(* IEC 61131-3 sources: elnaProjects/ElpcLogic/PomarKc7Changed/build_USO_ecl/_ (part 6) *)

  StrAlg.CanRun := StrAlg.inCanRun;
  StrAlg.OpcCommandsDisabled := StrAlg.inOpcCommandsDisabled;

  IF StrAlg.isRuning THEN

      StrAlg.hasError := kran3bOpen.error OR kran4Open.error OR kran5Close.error OR kran5Close.error
      OR kran1Open.error OR kran2Open.error OR kran3bClose.error OR kran4Close.error OR testUnsuccessfulFilling.error;

      IF kran4Open.top THEN
          runPhase(waitAfterKran4);
      END_IF;

      IF waitAfterKran4.top THEN
          runPhase(kran5Close);
      END_IF;

      IF kran3bOpen.top AND kran5Close.top THEN
         runPhase(waitAfterKran5);
         runPhase(didPKran1);
      END_IF;

      (*IF didPKran1.start AND NOT didPKran1.top THEN
      didPKran1.top:= im.singleSignals.dP_gazgaz_Kran1.Q;
      END_IF;*)

      IF waitAfterKran5.top AND didPKran1.top THEN
            runPhase(kran1Open);
  	runPhase(kran2Open);
      END_IF;

      IF kran1Open.top AND kran2Open.top THEN
            runPhase(kran4Close);
  	runPhase(kran3bClose);
      END_IF;

      IF kran4Close.top AND kran3bClose.top THEN

            runPhase(RunProtection_kr1);
            runPhase(RunProtection_kr2);

            (*runAiProtection(protections.Pgaza_na_vhode_nagnetatelia);
            runAiProtection(protections.Pgaza_na_vhode_nagnetatelia);
            runAiProtection(protections.Pgaza_na_vyhode_nagnetatelia);
            runAiProtection(protections.dPmaslo_gaz);
            runAiProtection(protections.Pmaslo_sm_nizkoe);
            runAiProtection(protections.Pmaslo_sm_vysokoe);*)

      END_IF;

      IF BreakPuskTimer.top AND NOT (RunProtection_kr1.top AND RunProtection_kr2.top ) THEN
  	testUnsuccessfulFilling.error:=TRUE;
      END_IF;

      IF RunProtection_kr1.top AND RunProtection_kr2.top THEN
            resetPhase(BreakPuskTimer);
  	waitReset(IN:=TRUE, PT:= T#2S);
      END_IF;

      IF waitReset.Q AND NOT (algoritms.Apusk.isRuning OR algoritms.SemiAutoPusk.isRuning) THEN
  	resetIfRunning(StrAlg);
      END_IF;

      StrAlg.isEnded:= RunProtection_kr1.top AND RunProtection_kr2.top;
  END_IF;

  StrAlg.CanRun := StrAlg.inCanRun;
  StrAlg.OpcCommandsDisabled := StrAlg.inOpcCommandsDisabled;

  (* ---- Если управление с ВУ заблокировано, то  передаем команду из алгоритма ---- *)
  IF StrAlg.inOpcCommandsDisabled THEN
  	StrAlg.inCommand := StrAlg.inCommand_Alg;
  ELSE (* иначе передаем команду с АРМа*)
  	StrAlg.inCommand := StrAlg.inCommand_ARM;
  END_IF;

  _sunpackerCommand(command := StrAlg.inCommand);
  	source := _sunpackerCommand.source;
  	cmd := _sunpackerCommand.cmd;

  IF cmd <> 0 AND lastCmd <> cmd AND (((NOT StrAlg.opcCommandsDisabled) AND source > 0) OR source = 0) then
  	CASE BYTE_TO_INT(cmd) OF
  		(*cmdRun*) 1: 	IF (StrAlg.CanRun) THEN
  					StrAlg.isRuning := TRUE;
  					StrAlg.isEnded := FALSE;
  					StrAlg.hasError := FALSE;
  					(*****************       OnRun       *****************)

                                                    runPhase(kran3bOpen);
                                                    runPhase(kran4Open);
                                                    runPhase(BreakPuskTimer);
                                                    runPhase(testUnsuccessfulFilling);

  					cmd_for_Status := cmd;
  					source_for_Status := source;
  					command_error_for_Status := 0;
  				ELSE
  					StrAlg.isRuning := FALSE;
  					StrAlg.isEnded := FALSE;
  					StrAlg.hasError 	:= FALSE;

  					cmd_for_Status := 0;
  					source_for_Status := source;
  					command_error_for_Status := cmd;
  				END_IF;
  		(*cmdReset*) 2: 	StrAlg.isRuning := FALSE;
  				StrAlg.isEnded := FALSE;
  				StrAlg.hasError 	:= FALSE;

                                           (*****************       OnReset       *****************)
                                          StrAlg.inCanRun:=FALSE;
                                          waitReset(IN:=FALSE);

                                          resetPhase(BreakPuskTimer);
                                          resetPhase(kran3bOpen);
                                          resetPhase(kran4Open);
                                          resetPhase(waitAfterKran4);
                                          resetPhase(kran5Close);
                                          resetPhase(didPKran1);
                                          resetPhase(kran1Open);
                                          resetPhase(kran2Open);
                                          resetPhase(kran3bClose);
                                          resetPhase(kran4Close);
  	                              resetPhase(RunProtection_kr1);
                                          resetPhase(RunProtection_kr2);
                                          resetPhase(waitAfterKran5);
                                          resetPhase(testUnsuccessfulFilling);

  				cmd_for_Status := cmd;
  				source_for_Status := source;
  				command_error_for_Status := 0;
  	END_CASE;
  	resetCmdTimer(IN := false);
  	resetCmdTimerPriznak := TRUE;
  END_IF;
  lastCmd := cmd;

  resetCmdTimer(IN := resetCmdTimerPriznak, PT := T#5S);
  IF resetCmdTimer.Q THEN
  	resetCmdTimerPriznak := FALSE;
  	source_for_Status := 0;
  	cmd_for_Status := 0;
  	command_error_for_Status := 0;
  END_IF;

  StrAlg.Start:= BreakPuskTimer.startStatus
              OR kran3bOpen.startStatus
              OR kran4Open.startStatus
              OR waitAfterKran4.startStatus
              OR kran5Close.startStatus
              OR didPKran1.startStatus
              OR kran1Open.startStatus
              OR kran2Open.startStatus
              OR kran3bClose.startStatus
              OR kran4Close.startStatus
              OR RunProtection_kr1.startStatus
              OR RunProtection_kr2.startStatus
              OR waitAfterKran5.startStatus
              OR testUnsuccessfulFilling.startStatus;

  StrAlg.Error:= BreakPuskTimer.errorStatus
              OR kran3bOpen.errorStatus
              OR kran4Open.errorStatus
              OR waitAfterKran4.errorStatus
              OR kran5Close.errorStatus
              OR didPKran1.errorStatus
              OR kran1Open.errorStatus
              OR kran2Open.errorStatus
              OR kran3bClose.errorStatus
              OR kran4Close.errorStatus
              OR RunProtection_kr1.errorStatus
              OR RunProtection_kr2.errorStatus
              OR waitAfterKran5.errorStatus
              OR testUnsuccessfulFilling.errorStatus;

  StrAlg.Top:=   BreakPuskTimer.topStatus
              OR kran3bOpen.topStatus
              OR kran4Open.topStatus
              OR waitAfterKran4.topStatus
              OR kran5Close.topStatus
              OR didPKran1.topStatus
              OR kran1Open.topStatus
              OR kran2Open.topStatus
              OR kran3bClose.topStatus
              OR kran4Close.topStatus
              OR RunProtection_kr1.topStatus
              OR RunProtection_kr2.topStatus
              OR waitAfterKran5.topStatus
              OR testUnsuccessfulFilling.topStatus;

  (*TODO: TYPE PROGRAM CODE HERE*)
  StrAlg.status :=  SHL(BYTE_TO_DWORD(source_for_Status), 29)
  			OR SHL(BYTE_TO_DWORD(cmd_for_Status), 26)
  			OR SHL(BYTE_TO_DWORD(command_error_for_Status), 23)
  			OR SHL(BOOL_TO_DWORD(StrAlg.OpcCommandsDisabled ), 21)
  			OR SHL(BOOL_TO_DWORD(StrAlg.hasError),4)
  			OR SHL(BOOL_TO_DWORD(StrAlg.CanRun),2)
  			OR SHL(BOOL_TO_DWORD(StrAlg.isEnded),1)
  			OR BOOL_TO_DWORD(StrAlg.isRuning);
END_FUNCTION_BLOCK

FUNCTION_BLOCK engineRunAlg
  VAR_IN_OUT
    StrAlg : struct_Alg;
  END_VAR
  VAR
    BreakPuskTimer : struct_PhaseAlgoritm;
    RunProtection_mvoff : struct_PhaseAlgoritm;
    LowOil_upStopust : struct_PhaseAlgoritm;
    mvOn : struct_PhaseAlgoritm;
    AutoPns_ph : struct_PhaseAlgoritm;
    AutoAvom_ph : struct_PhaseAlgoritm;
    pnsOff : struct_PhaseAlgoritm;
    testUnsuccessful : struct_PhaseAlgoritm;
    fb_BreakPuskTimer : fb_ph_Timer;
    fb_RunProtection_mvoff : fb_ph_DIprotection;
    fb_LowOil_upStopust : fb_ph_WaitAnalogValue;
    fb_mvOn : fb_ph_SectionSwitch;
    fb_AutoPns_ph : fb_ph_algoritm;
    fb_AutoAvom_ph : fb_ph_algoritm;
    fb_pnsOff : fb_ph_Switch;
    fb_testUnsuccessful : fb_ph_CustomPhase;
    _sunpackerCommand : fb_sunpackerCommand;
    _DualStateImAction : TYPE_DualStateImAction;
    _PhaseAlgoritmAction : TYPE_PhaseAlgoritmAction;
    source : BYTE;
    cmd : BYTE;
    lastCmd : BYTE;
    source_for_Status : BYTE;
    cmd_for_Status : BYTE;
    command_error_for_Status : BYTE;
    resetCmdTimer : TON;
    resetCmdTimerPriznak : BOOL;
    onInit : BOOL;
    waitReset : TON;
  END_VAR
  VAR_EXTERNAL
    IM : ImConfig;
    algoritms : AlgoritmsConfig;
    ai : AiConfig;
    protections : ProtectionsConfig;
    AlgTimers : struct_AlgTimers;
  END_VAR

  IF NOT onInit THEN

       fb_BreakPuskTimer(phaseNumber:=0, delay:=T#665S);
     fb_LowOil_upStopust(phaseNumber:=1);
                 fb_mvOn(phaseNumber:=2, act:=_on);
           fb_AutoPns_ph(phaseNumber:=3, act:=_run, waitCompletion:=FALSE);
          fb_AutoAvom_ph(phaseNumber:=4, act:=_run, waitCompletion:=FALSE);
               fb_pnsOff(phaseNumber:=5, act:=_off);
  fb_RunProtection_mvoff(phaseNumber:=7, act:=_run);
     fb_testUnsuccessful(phaseNumber:=17);

  onInit:=TRUE;
  END_IF;

          fb_BreakPuskTimer(StrPh:=BreakPuskTimer, timer:=AlgTimers.engineRun_BreakPuskTimer);
       (* fb_LowOil_upStopust(StrPh:=LowOil_upStopust, ai:=ai.Pmasla_posle_GNS, more:=im.AutoPns_UstStop.Value);*)
                    fb_mvOn(StrPh:=mvOn, Im:=Im.mv);
              fb_AutoPns_ph(StrPh:=AutoPns_ph, alg:=algoritms.AutoPns);
             fb_AutoAvom_ph(StrPh:=AutoAvom_ph, alg:=algoritms.AutoAvom);
                  fb_pnsOff(StrPh:=pnsOff, Im:=Im.pns);
    (*fb_RunProtection_mvoff(StrPh:=RunProtection_mvoff, StrDiP:=protections.Pgaza_na_vyhode_nagnetatelia_GPA_STOP);*)
        fb_testUnsuccessful(StrPh:=testUnsuccessful);

  StrAlg.CanRun := StrAlg.inCanRun;
  StrAlg.OpcCommandsDisabled := StrAlg.inOpcCommandsDisabled;

  IF StrAlg.isRuning THEN

      StrAlg.hasError := mvOn.error OR pnsOff.error OR testUnsuccessful.error;

      IF mvOn.top THEN
          runPhase(RunProtection_mvoff);
          runPhase(AutoAvom_ph);
          runPhase(LowOil_upStopust);
      END_IF;
      (*
      IF AutoAvom_ph.top THEN
          algoritms.AutoAvom.inOpcCommandsDisabled:=FALSE;
      END_IF;
      *)
      IF LowOil_upStopust.top THEN
          runPhase(pnsOff);
      END_IF;

      IF pnsOff.top THEN
         runPhase(AutoPns_ph);
      END_IF;

      IF BreakPuskTimer.top AND NOT AutoPns_ph.top THEN
            testUnsuccessful.error:=TRUE;
      END_IF;

      IF AutoPns_ph.top THEN
            resetPhase(BreakPuskTimer);
  	waitReset(IN:=TRUE, PT:= T#2S);
      END_IF;

      IF waitReset.Q AND NOT (algoritms.Apusk.isRuning OR algoritms.SemiAutoPusk.isRuning) THEN
  	resetIfRunning(StrAlg);
      END_IF;

      StrAlg.isEnded:= AutoPns_ph.top;
  END_IF;

  StrAlg.CanRun := StrAlg.inCanRun;
  StrAlg.OpcCommandsDisabled := StrAlg.inOpcCommandsDisabled;

  (* ---- Если управление с ВУ заблокировано, то  передаем команду из алгоритма ---- *)
  IF StrAlg.inOpcCommandsDisabled THEN
  	StrAlg.inCommand := StrAlg.inCommand_Alg;
  ELSE (* иначе передаем команду с АРМа*)
  	StrAlg.inCommand := StrAlg.inCommand_ARM;
  END_IF;

  _sunpackerCommand(command := StrAlg.inCommand);
  	source := _sunpackerCommand.source;
  	cmd := _sunpackerCommand.cmd;

  IF cmd <> 0 AND lastCmd <> cmd AND (((NOT StrAlg.opcCommandsDisabled) AND source > 0) OR source = 0) then
  	CASE BYTE_TO_INT(cmd) OF
  		(*cmdRun*) 1: 	IF (StrAlg.CanRun) THEN
  					StrAlg.isRuning := TRUE;
  					StrAlg.isEnded := FALSE;
  					StrAlg.hasError := FALSE;
  					(*****************       OnRun       *****************)

                                                    runPhase(mvOn);
                                                    runPhase(BreakPuskTimer);
                                                    runPhase(testUnsuccessful);

  					cmd_for_Status := cmd;
  					source_for_Status := source;
  					command_error_for_Status := 0;
  				ELSE
  					StrAlg.isRuning := FALSE;
  					StrAlg.isEnded := FALSE;
  					StrAlg.hasError 	:= FALSE;

  					cmd_for_Status := 0;
  					source_for_Status := source;
  					command_error_for_Status := cmd;
  				END_IF;
  		(*cmdReset*) 2: 	StrAlg.isRuning := FALSE;
  				StrAlg.isEnded := FALSE;
  				StrAlg.hasError 	:= FALSE;

                                           (*****************       OnReset       *****************)
                                          StrAlg.inCanRun:=FALSE;
                                          waitReset(IN:=FALSE);

                                          resetPhase(BreakPuskTimer);
                                          resetPhase(RunProtection_mvoff);
                                          resetPhase(LowOil_upStopust);
                                          resetPhase(mvOn);
                                          resetPhase(AutoPns_ph);
                                          resetPhase(AutoAvom_ph);
                                          resetPhase(pnsOff);
                                          resetPhase(testUnsuccessful);

  				cmd_for_Status := cmd;
  				source_for_Status := source;
  				command_error_for_Status := 0;
  	END_CASE;
  	resetCmdTimer(IN := false);
  	resetCmdTimerPriznak := TRUE;
  END_IF;
  lastCmd := cmd;

  resetCmdTimer(IN := resetCmdTimerPriznak, PT := T#5S);
  IF resetCmdTimer.Q THEN
  	resetCmdTimerPriznak := FALSE;
  	source_for_Status := 0;
  	cmd_for_Status := 0;
  	command_error_for_Status := 0;
  END_IF;

  StrAlg.Start:= BreakPuskTimer.startStatus
              OR RunProtection_mvoff.startStatus
              OR LowOil_upStopust.startStatus
              OR mvOn.startStatus
              OR AutoPns_ph.startStatus
              OR AutoAvom_ph.startStatus
              OR pnsOff.startStatus
              OR testUnsuccessful.startStatus;

  StrAlg.Error:= BreakPuskTimer.errorStatus
              OR RunProtection_mvoff.errorStatus
              OR LowOil_upStopust.errorStatus
              OR mvOn.errorStatus
              OR AutoPns_ph.errorStatus
              OR AutoAvom_ph.errorStatus
              OR pnsOff.errorStatus
              OR testUnsuccessful.errorStatus;

  StrAlg.Top:=   BreakPuskTimer.topStatus
              OR RunProtection_mvoff.topStatus
              OR LowOil_upStopust.topStatus
              OR mvOn.topStatus
              OR AutoPns_ph.topStatus
              OR AutoAvom_ph.topStatus
              OR pnsOff.topStatus
              OR testUnsuccessful.topStatus;

  (*TODO: TYPE PROGRAM CODE HERE*)
  StrAlg.status :=  SHL(BYTE_TO_DWORD(source_for_Status), 29)
  			OR SHL(BYTE_TO_DWORD(cmd_for_Status), 26)
  			OR SHL(BYTE_TO_DWORD(command_error_for_Status), 23)
  			OR SHL(BOOL_TO_DWORD(StrAlg.OpcCommandsDisabled ), 21)
  			OR SHL(BOOL_TO_DWORD(StrAlg.hasError),4)
  			OR SHL(BOOL_TO_DWORD(StrAlg.CanRun),2)
  			OR SHL(BOOL_TO_DWORD(StrAlg.isEnded),1)
  			OR BOOL_TO_DWORD(StrAlg.isRuning);
END_FUNCTION_BLOCK

FUNCTION_BLOCK puskKalg
  VAR_IN_OUT
    StrAlg : struct_Alg;
  END_VAR
  VAR
    puskOilSystem : struct_PhaseAlgoritm;
  END_VAR
  VAR_IN_OUT
    questionFilling : struct_Question;
  END_VAR
  VAR
    filling : struct_PhaseAlgoritm;
  END_VAR
  VAR_IN_OUT
    questionUnload : struct_Question;
  END_VAR
  VAR
    kran3bOpen : struct_PhaseAlgoritm;
    kran4Close : struct_PhaseAlgoritm;
    kran1Close : struct_PhaseAlgoritm;
    kran2Close : struct_PhaseAlgoritm;
    kran5open : struct_PhaseAlgoritm;
    wait720 : struct_PhaseAlgoritm;
    noGasInPipe : struct_PhaseAlgoritm;
    AutoNUoff : struct_PhaseAlgoritm;
    nu1Off : struct_PhaseAlgoritm;
    nu2Off : struct_PhaseAlgoritm;
    pnsWaitOff : struct_PhaseAlgoritm;
    testUnsuccessfulUnfill : struct_PhaseAlgoritm;
    fb_puskOilSystem : fb_ph_algoritm;
    fb_questionFilling : fb_Question;
    fb_filling : fb_ph_algoritm;
    fb_questionUnload : fb_Question;
    fb_kran3bOpen : fb_ph_Kran;
    fb_kran4Close : fb_ph_CustomPhase;
    fb_kran1Close : fb_ph_Kran;
    fb_kran2Close : fb_ph_Kran;
    fb_kran5open : fb_ph_Kran;
    fb_wait720 : fb_ph_Timer;
    fb_noGasInPipe : fb_ph_CustomPhase;
    fb_AutoNUoff : fb_ph_algoritm;
    fb_nu1Off : fb_ph_OilPump;
    fb_nu2Off : fb_ph_OilPump;
    fb_pnsWaitOff : fb_ph_algoritm;
    fb_testUnsuccessfulUnfill : fb_ph_CustomPhase;
    _sunpackerCommand : fb_sunpackerCommand;
    _DualStateImAction : TYPE_DualStateImAction;
    _Answers : TYPE_Answers;
    _statusDualInput : TYPE_statusDualInput;
    _StatusAi : TYPE_StatusAi;
    _PhaseAlgoritmAction : TYPE_PhaseAlgoritmAction;
    source : BYTE;
    cmd : BYTE;
    lastCmd : BYTE;
    source_for_Status : BYTE;
    cmd_for_Status : BYTE;
    command_error_for_Status : BYTE;
    resetCmdTimer : TON;
    resetCmdTimerPriznak : BOOL;
    OpcCommandsKransEnabled : BOOL;
    OpcCommandsKransDisabled : BOOL;
    _resetQuestion1 : BOOL;
    _resetQuestion2 : BOOL;
    onInit : BOOL;
    waitReset : TON;
  END_VAR
  VAR_EXTERNAL
    IM : ImConfig;
    algoritms : AlgoritmsConfig;
    ai : AiConfig;
    AlgTimers : struct_AlgTimers;
    ModeGpa : TYPE_ModeGpa;
    algManager : struct_AlgoritmsManager;
    protections : ProtectionsConfig;
  END_VAR
  VAR CONSTANT
    Ust_Pgaza : LREAL      := 0.3;
  END_VAR

  IF NOT onInit THEN

            fb_puskOilSystem(phaseNumber:=0, act:=_run, waitCompletion:=TRUE);
        questionFilling.AnswerVariants:=_Answers.ANS_YES;
                  fb_filling(phaseNumber:=1, act:=_run, waitCompletion:=TRUE);
      questionUnload.AnswerVariants:=_Answers.ANS_YES;
               fb_kran3bOpen(phaseNumber:=3, act:=_on);
               fb_kran4Close(phaseNumber:=4);
               fb_kran1Close(phaseNumber:=5, act:=_off);
               fb_kran2Close(phaseNumber:=6, act:=_off);
                fb_kran5open(phaseNumber:=7, act:=_on);
                  fb_wait720(phaseNumber:=8, delay:=T#720S);
              fb_noGasInPipe(phaseNumber:=9);
                fb_AutoNUoff(phaseNumber:=10, act:=_reset, waitCompletion:=FALSE);
                   fb_nu1Off(phaseNumber:=11, act:=_off);
                   fb_nu2Off(phaseNumber:=12, act:=_off);
               fb_pnsWaitOff(phaseNumber:=15, act:=_run, waitCompletion:=TRUE);
   fb_testUnsuccessfulUnfill(phaseNumber:=18);

  onInit:=TRUE;
  END_IF;

            fb_puskOilSystem(StrPh:=puskOilSystem, alg:=algoritms.puskOilSystem);
          fb_questionFilling(StrQ:=questionFilling);
                  fb_filling(StrPh:=filling, alg:=algoritms.filling);
           fb_questionUnload(StrQ:=questionUnload);
               fb_kran3bOpen(StrPh:=kran3bOpen, Im:=Im.kran3b);
               fb_kran4Close(StrPh:=kran4Close);
               fb_kran1Close(StrPh:=kran1Close, Im:=Im.kran1);
               fb_kran2Close(StrPh:=kran2Close, Im:=Im.kran2);
                fb_kran5open(StrPh:=kran5open, Im:=Im.kran5);
                  fb_wait720(StrPh:=wait720, timer:=AlgTimers.puskK_wait720);
              fb_noGasInPipe(StrPh:=noGasInPipe);
                fb_AutoNUoff(StrPh:=AutoNUoff, alg:=algoritms.autoNu);
                   fb_nu1Off(StrPh:=nu1Off, Im:=Im.nu1);
                   fb_nu2Off(StrPh:=nu2Off, Im:=Im.nu2);
               fb_pnsWaitOff(StrPh:=pnsWaitOff, alg:=algoritms.vibegPNS);
   fb_testUnsuccessfulUnfill(StrPh:=testUnsuccessfulUnfill);

  StrAlg.CanRun := StrAlg.inCanRun;
  StrAlg.OpcCommandsDisabled := StrAlg.inOpcCommandsDisabled;

  IF StrAlg.isRuning THEN

      StrAlg.hasError := kran3bOpen.error OR kran1Close.error OR kran2Close.error OR kran5open.error OR testUnsuccessfulUnfill.error;

      IF puskOilSystem.top THEN
           IF NOT _resetQuestion1 THEN
           askQuestion(questionFilling);
           _resetQuestion1:=TRUE;
           END_IF;
      END_IF;

      IF questionFilling.answer = _Answers.ANS_YES THEN
          runPhase(filling);
          resetQuestion(questionFilling);
      END_IF;

      IF filling.top THEN
         OpcCommandsKransEnabled:=TRUE;
         resetDiProtection(protections.Reg_vozb_off);
         (*resetDiProtection(protections.Fail_chastotnii_pusk);*)
         IF NOT _resetQuestion2 THEN
         askQuestion(questionUnload);
         _resetQuestion2:=TRUE;
         END_IF;
      END_IF;

       IF questionUnload.answer = _Answers.ANS_YES THEN
          OpcCommandsKransDisabled:=TRUE;
          runPhase(kran3bOpen);
          runPhase(wait720);
          resetQuestion(questionUnload);
      END_IF;

      IF kran3bOpen.top THEN
            resetDiProtection(protections.Reg_vozb_off);
            resetDiProtection(protections.Fail_chastotnii_pusk);

            runPhase(kran1Close);
            runPhase(kran2Close);
            runPhase(kran4Close);
      END_IF;

       IF kran4Close.start AND NOT kran4Close.top THEN
  	kran4Close.top:= Im.kran4.onStatus = _statusDualInput.STATUS_OFF;
      END_IF;

      IF kran1Close.top AND kran2Close.top AND kran4Close.top THEN
  	runPhase(kran5open);
      END_IF;

      IF kran5open.top THEN
  	runPhase(noGasInPipe);
      END_IF;

      IF noGasInPipe.start AND (NOT noGasInPipe.top) THEN
  	noGasInPipe.top:=  (ai.dPgaza_na_maslo_filtre.interval >= _statusAi.NORMAL
                           AND  ai.dPgaza_na_maslo_filtre.value< Ust_Pgaza )
                           AND (ai.Pmaslo_sm_vysokoe.interval >= _statusAi.NORMAL
                           AND  ai.Pmaslo_sm_vysokoe.value< Ust_Pgaza);
      END_IF;

      IF noGasInPipe.top THEN

            ai.Tmasla_MB.Disabled_LA:=TRUE;
            ai.Tmasla_MB.Disabled_LW:=TRUE;
            (*IM.SingleSignals.dP_oilgaz_low.Disabled_Sig:=TRUE;*)
            resetAiProtection(protections.Os_sdvig_nagnetatelja_plus);
           (* resetDiProtection(protections.Vibro_skorost_OP_shesterni_RED_T5);*)
  	runPhase(AutoNUoff);

      END_IF;

       IF autoNuOff.top THEN
  	runPhase(nu1off);
            runPhase(nu2off);
      END_IF;

      IF nu1Off.top AND nu2Off.top THEN
  	runPhase(pnsWaitOff);
      END_IF;

      IF wait720.top AND NOT (pnsWaitOff.top) THEN
            testUnsuccessfulUnfill.error:=TRUE;
      END_IF;

      IF pnsWaitOff.top THEN
            resetPhase(wait720);
  	waitReset(IN:=TRUE, PT:= T#3S);
      END_IF;

      IF waitReset.Q THEN
          resetIfRunning(algoritms.vibegPNS);
          algManager.nMode:=ModeGpa.MODE_STOP;
          resetIfRunning(StrAlg);
      END_IF;

      StrAlg.isEnded:= pnsWaitOff.top;

      IF OpcCommandsKransEnabled AND NOT OpcCommandsKransDisabled THEN
  	IF      (im.pns.onStatus = _statusDualInput.STATUS_ON)
                AND (im.nu1.onStatus = _statusDualInput.STATUS_ON OR im.nu2.onStatus = _statusDualInput.STATUS_ON)
  	    AND (ai.Tmasla_MB.interval >= _statusAi.normal)
                (*AND (ai.Tmasla_MB.value > im.PuskOilSystem_UstdPmg.Value)*)
            THEN
  	    IM.Kran3b.inOpcCommandsDisabled:=FALSE;
  	    Im.kran4.inOpcCommandsDisabled:=FALSE;
  	    Im.kran5.inOpcCommandsDisabled:=FALSE;
  		(*IF	Im.SingleSignals.dP_gazgaz_Kran1.q THEN
  			Im.kran1.inOpcCommandsDisabled:=FALSE;
  			Im.kran2.inOpcCommandsDisabled:=FALSE;
  		ELSE
  			Im.kran1.inOpcCommandsDisabled:=TRUE;
  			Im.kran2.inOpcCommandsDisabled:=TRUE;
  		END_IF;*)
            ELSE
  	    Im.kran1.inOpcCommandsDisabled:=TRUE;
  	    Im.kran2.inOpcCommandsDisabled:=TRUE;
  	    Im.kran3b.inOpcCommandsDisabled:=TRUE;
  	    Im.kran4.inOpcCommandsDisabled:=TRUE;
  	    Im.kran5.inOpcCommandsDisabled:=TRUE;
            END_IF;

      ELSE
  	Im.kran1.inOpcCommandsDisabled:=TRUE;
  	Im.kran2.inOpcCommandsDisabled:=TRUE;
  	Im.kran3b.inOpcCommandsDisabled:=TRUE;
  	Im.kran4.inOpcCommandsDisabled:=TRUE;
  	Im.kran5.inOpcCommandsDisabled:=TRUE;
      END_IF;
  END_IF;

  StrAlg.CanRun := StrAlg.inCanRun;
  StrAlg.OpcCommandsDisabled := StrAlg.inOpcCommandsDisabled;

  (* ---- Если управление с ВУ заблокировано, то  передаем команду из алгоритма ---- *)
  IF StrAlg.inOpcCommandsDisabled THEN
  	StrAlg.inCommand := StrAlg.inCommand_Alg;
  ELSE (* иначе передаем команду с АРМа*)
  	StrAlg.inCommand := StrAlg.inCommand_ARM;
  END_IF;

  _sunpackerCommand(command := StrAlg.inCommand);
  	source := _sunpackerCommand.source;
  	cmd := _sunpackerCommand.cmd;

  IF cmd <> 0 AND lastCmd <> cmd AND (((NOT StrAlg.opcCommandsDisabled) AND source > 0) OR source = 0) then
  	CASE BYTE_TO_INT(cmd) OF
  		(*cmdRun*) 1: 	IF (StrAlg.CanRun) THEN
  					StrAlg.isRuning := TRUE;
  					StrAlg.isEnded := FALSE;
  					StrAlg.hasError := FALSE;
  					(*****************       OnRun       *****************)

                                                    algManager.nMode:=ModeGpa.MODE_PUSKK;
                                                    resetAndDisable(alg:=algoritms.ppu);
                                                    algoritms.puskOilSystem.inCanRun:= TRUE;
                                                    algoritms.filling.inCanRun:= TRUE;
                                                    runPhase(puskOilSystem);

  					cmd_for_Status := cmd;
  					source_for_Status := source;
  					command_error_for_Status := 0;
  				ELSE
  					StrAlg.isRuning := FALSE;
  					StrAlg.isEnded := FALSE;
  					StrAlg.hasError 	:= FALSE;

  					cmd_for_Status := 0;
  					source_for_Status := source;
  					command_error_for_Status := cmd;
  				END_IF;
  		(*cmdReset*) 2: 	StrAlg.isRuning := FALSE;
  				StrAlg.isEnded := FALSE;
  				StrAlg.hasError 	:= FALSE;

                                           (*****************       OnReset       *****************)
                                          OpcCommandsKransEnabled:=FALSE;
                                          OpcCommandsKransDisabled:=FALSE;
                                          waitReset(IN:=FALSE);
                                          _resetQuestion1:=FALSE;
                                          _resetQuestion2:=FALSE;
                                          resetPhase(puskOilSystem);
                                          resetPhase(filling);
                                          resetPhase(kran3bOpen);
                                          resetPhase(kran4Close);
                                          resetPhase(kran1Close);
                                          resetPhase(kran2Close);
                                          resetPhase(kran5open);
                                          resetPhase(wait720);
                                          resetPhase(noGasInPipe);
                                          resetPhase(AutoNUoff);
                                          resetPhase(nu1Off);
                                          resetPhase(nu2Off);
                                          resetPhase(pnsWaitOff);
                                          resetPhase(testUnsuccessfulUnfill);
                                          BlockAllIM(IM);
                                          resetQuestion(questionFilling);
                                          resetQuestion(questionUnload);

                                          StrAlg.inOpcCommandsDisabled:=FALSE;

  				cmd_for_Status := cmd;
  				source_for_Status := source;
  				command_error_for_Status := 0;
  	END_CASE;
  	resetCmdTimer(IN := false);
  	resetCmdTimerPriznak := TRUE;
  END_IF;
  lastCmd := cmd;

  resetCmdTimer(IN := resetCmdTimerPriznak, PT := T#5S);
  IF resetCmdTimer.Q THEN
  	resetCmdTimerPriznak := FALSE;
  	source_for_Status := 0;
  	cmd_for_Status := 0;
  	command_error_for_Status := 0;
  END_IF;

  StrAlg.Start:= puskOilSystem.startStatus
              OR filling.startStatus
              OR kran3bOpen.startStatus
              OR kran4Close.startStatus
              OR kran1Close.startStatus
              OR kran2Close.startStatus
              OR kran5open.startStatus
              OR wait720.startStatus
              OR noGasInPipe.startStatus
              OR AutoNUoff.startStatus
              OR nu1Off.startStatus
              OR nu2Off.startStatus
              OR pnsWaitOff.startStatus
              OR testUnsuccessfulUnfill.startStatus;

  StrAlg.Error:=  puskOilSystem.errorStatus
              OR filling.errorStatus
              OR kran3bOpen.errorStatus
              OR kran4Close.errorStatus
              OR kran1Close.errorStatus
              OR kran2Close.errorStatus
              OR kran5open.errorStatus
              OR wait720.errorStatus
              OR noGasInPipe.errorStatus
              OR AutoNUoff.errorStatus
              OR nu1Off.errorStatus
              OR nu2Off.errorStatus
              OR pnsWaitOff.errorStatus
              OR testUnsuccessfulUnfill.errorStatus;

  StrAlg.Top:=   puskOilSystem.topStatus
              OR filling.topStatus
              OR kran3bOpen.topStatus
              OR kran4Close.topStatus
              OR kran1Close.topStatus
              OR kran2Close.topStatus
              OR kran5open.topStatus
              OR wait720.topStatus
              OR noGasInPipe.topStatus
              OR AutoNUoff.topStatus
              OR nu1Off.topStatus
              OR nu2Off.topStatus
              OR pnsWaitOff.topStatus
              OR testUnsuccessfulUnfill.topStatus;

  (*TODO: TYPE PROGRAM CODE HERE*)
  StrAlg.status :=  SHL(BYTE_TO_DWORD(source_for_Status), 29)
  			OR SHL(BYTE_TO_DWORD(cmd_for_Status), 26)
  			OR SHL(BYTE_TO_DWORD(command_error_for_Status), 23)
  			OR SHL(BOOL_TO_DWORD(StrAlg.OpcCommandsDisabled ), 21)
  			OR SHL(BOOL_TO_DWORD(StrAlg.hasError),4)
  			OR SHL(BOOL_TO_DWORD(StrAlg.CanRun),2)
  			OR SHL(BOOL_TO_DWORD(StrAlg.isEnded),1)
  			OR BOOL_TO_DWORD(StrAlg.isRuning);
END_FUNCTION_BLOCK

FUNCTION_BLOCK puskValg
  VAR_IN_OUT
    StrAlg : struct_Alg;
  END_VAR
  VAR
    puskOilSystem : struct_PhaseAlgoritm;
  END_VAR
  VAR_IN_OUT
    questionEngine : struct_Question;
  END_VAR
  VAR
    runningEngine : struct_PhaseAlgoritm;
  END_VAR
  VAR_IN_OUT
    questionMVoff : struct_Question;
  END_VAR
  VAR
    mvOff : struct_PhaseAlgoritm;
    pnsOn : struct_PhaseAlgoritm;
    wait600 : struct_PhaseAlgoritm;
    AutoNUoff : struct_PhaseAlgoritm;
    nu1Off : struct_PhaseAlgoritm;
    nu2Off : struct_PhaseAlgoritm;
    autoAvomOff : struct_PhaseAlgoritm;
    Avom1Off : struct_PhaseAlgoritm;
    Avom2Off : struct_PhaseAlgoritm;
    pnsWaitOff : struct_PhaseAlgoritm;
    testUnsuccessful : struct_PhaseAlgoritm;
    fb_puskOilSystem : fb_ph_algoritm;
    fb_questionEngine : fb_Question;
    fb_runningEngine : fb_ph_algoritm;
    fb_questionMVoff : fb_Question;
    fb_mvOff : fb_ph_SectionSwitch;
    fb_pnsOn : fb_ph_Switch;
    fb_wait600 : fb_ph_Timer;
    fb_AutoNUoff : fb_ph_algoritm;
    fb_nu1Off : fb_ph_OilPump;
    fb_nu2Off : fb_ph_OilPump;
    fb_autoAvomOff : fb_ph_algoritm;
    fb_Avom1Off : fb_ph_Switch;
    fb_Avom2Off : fb_ph_Switch;
    fb_pnsWaitOff : fb_ph_algoritm;
    fb_testUnsuccessful : fb_ph_CustomPhase;
    _sunpackerCommand : fb_sunpackerCommand;
    _DualStateImAction : TYPE_DualStateImAction;
    _Answers : TYPE_Answers;
    _statusDualInput : TYPE_statusDualInput;
    _StatusAi : TYPE_StatusAi;
    _PhaseAlgoritmAction : TYPE_PhaseAlgoritmAction;
    source : BYTE;
    cmd : BYTE;
    lastCmd : BYTE;
    source_for_Status : BYTE;
    cmd_for_Status : BYTE;
    command_error_for_Status : BYTE;
    resetCmdTimer : TON;
    resetCmdTimerPriznak : BOOL;
    onInit : BOOL;
    _resetQuestion1 : BOOL;
    _resetQuestion2 : BOOL;
    waitReset : TON;
  END_VAR
  VAR_EXTERNAL
    IM : ImConfig;
    algoritms : AlgoritmsConfig;
    ai : AiConfig;
    AlgTimers : struct_AlgTimers;
    ModeGpa : TYPE_ModeGpa;
    algManager : struct_AlgoritmsManager;
    protections : ProtectionsConfig;
  END_VAR
  VAR CONSTANT
    Ust_Pgaza : LREAL      := 0.3;
  END_VAR

  IF NOT onInit THEN

            fb_puskOilSystem(phaseNumber:=0, act:=_run, waitCompletion:=TRUE);
         questionEngine.AnswerVariants:=_Answers.ANS_YES;
            fb_runningEngine(phaseNumber:=1, act:=_run, waitCompletion:=TRUE);
          questionMVoff.AnswerVariants:=_Answers.ANS_YES;
                    fb_mvOff(phaseNumber:=3, act:=_off);
                    fb_pnsOn(phaseNumber:=4, act:=_on);
                  fb_wait600(phaseNumber:=8, delay:=T#600S);
                fb_AutoNUoff(phaseNumber:=10, act:=_reset, waitCompletion:=FALSE);
                   fb_nu1Off(phaseNumber:=11, act:=_off);
                   fb_nu2Off(phaseNumber:=12, act:=_off);
               fb_pnsWaitOff(phaseNumber:=15, act:=_run, waitCompletion:=TRUE);
              fb_autoAvomOff(phaseNumber:=7, act:=_reset, waitCompletion:=FALSE);
                 fb_Avom1Off(phaseNumber:=5, act:=_off);
                 fb_Avom2Off(phaseNumber:=6, act:=_off);
         fb_testUnsuccessful(phaseNumber:=17);

  onInit:=TRUE;
  END_IF;

            fb_puskOilSystem(StrPh:=puskOilSystem, alg:=algoritms.puskOilSystem);
           fb_questionEngine(StrQ:=questionEngine);
            fb_runningEngine(StrPh:=runningEngine, alg:=algoritms.engineRun);
            fb_questionMVoff(StrQ:=questionMVoff);
                    fb_mvOff(StrPh:=mvOff, Im:=Im.mv);
                    fb_pnsOn(StrPh:=pnsOn, Im:=Im.pns);
                  fb_wait600(StrPh:=wait600, timer:=AlgTimers.puskV_wait600);
                fb_AutoNUoff(StrPh:=AutoNUoff, alg:=algoritms.autoNu);
                   fb_nu1Off(StrPh:=nu1Off, Im:=Im.nu1);
                   fb_nu2Off(StrPh:=nu2Off, Im:=Im.nu2);
               fb_pnsWaitOff(StrPh:=pnsWaitOff, alg:=algoritms.vibegPNS);
              fb_autoAvomOff(StrPh:=autoAvomOff, alg:=algoritms.AutoAvom);
                 fb_Avom1Off(StrPh:=Avom1Off, Im:=Im.v1_Avom);
                 fb_Avom2Off(StrPh:=Avom2Off, Im:=Im.v2_Avom);
         fb_testUnsuccessful(StrPh:=testUnsuccessful);

  StrAlg.CanRun := StrAlg.inCanRun;
  StrAlg.OpcCommandsDisabled := StrAlg.inOpcCommandsDisabled;

  IF StrAlg.isRuning THEN

      StrAlg.hasError := mvOff.error OR pnsOn.error OR testUnsuccessful.error;

      IF puskOilSystem.top THEN
           IF NOT _resetQuestion1 THEN
           askQuestion(questionEngine);
           _resetQuestion1:=TRUE;
           END_IF;
      END_IF;

      IF questionEngine.answer = _Answers.ANS_YES THEN
          runPhase(runningEngine);
          resetQuestion(questionEngine);
      END_IF;

      IF runningEngine.top THEN
         IF NOT _resetQuestion2 THEN
         askQuestion(questionMVoff);
         _resetQuestion2:=TRUE;
         END_IF;
      END_IF;

       IF questionMVoff.answer = _Answers.ANS_YES THEN

          (*resetDiProtection(protections.Pgaza_na_vyhode_nagnetatelia_GPA_STOP);
         *) resetIfRunning(algoritms.AutoPns);
          runPhase(mvOff);
          runPhase(wait600);
          resetQuestion(questionMVoff);
       END_IF;

      IF mvOff.top THEN
          runPhase(pnsOn);
      END_IF;

      IF pnsOn.top THEN

            ai.Tmasla_MB.Disabled_LA:=TRUE;
            ai.Tmasla_MB.Disabled_LW:=TRUE;
            (*IM.SingleSignals.dP_oilgaz_low.Disabled_Sig:=TRUE;*)
            (*resetAiProtection(protections.Os_sdvig_nagnetatelja_plus)*)
           (* resetDiProtection(protections.Vibro_skorost_OP_shesterni_RED_T5);*)
  	runPhase(AutoNUoff);

      END_IF;

       IF autoNuOff.top THEN
  	runPhase(nu1off);
            runPhase(nu2off);
      END_IF;

      IF nu1Off.top AND nu2Off.top THEN
  	runPhase(pnsWaitOff);
      END_IF;

      IF wait600.top AND NOT (pnsWaitOff.top) THEN
            testUnsuccessful.error:=TRUE;
      END_IF;

      IF pnsWaitOff.top THEN
            resetPhase(wait600);
            runPhase(autoAvomOff);
  	waitReset(IN:=TRUE, PT:= T#3S);
      END_IF;

      IF autoAvomOff.top THEN
            runPhase(Avom1Off);
            runPhase(Avom2Off);
      END_IF;

      IF waitReset.Q THEN
          resetIfRunning(algoritms.vibegPNS);
          algManager.nMode:=ModeGpa.MODE_STOP;
          resetIfRunning(StrAlg);
      END_IF;

      StrAlg.isEnded:= pnsWaitOff.top;

  END_IF;

  StrAlg.CanRun := StrAlg.inCanRun;
  StrAlg.OpcCommandsDisabled := StrAlg.inOpcCommandsDisabled;

  (* ---- Если управление с ВУ заблокировано, то  передаем команду из алгоритма ---- *)
  IF StrAlg.inOpcCommandsDisabled THEN
  	StrAlg.inCommand := StrAlg.inCommand_Alg;
  ELSE (* иначе передаем команду с АРМа*)
  	StrAlg.inCommand := StrAlg.inCommand_ARM;
  END_IF;

  _sunpackerCommand(command := StrAlg.inCommand);
  	source := _sunpackerCommand.source;
  	cmd := _sunpackerCommand.cmd;

  IF cmd <> 0 AND lastCmd <> cmd AND (((NOT StrAlg.opcCommandsDisabled) AND source > 0) OR source = 0) then
  	CASE BYTE_TO_INT(cmd) OF
  		(*cmdRun*) 1: 	IF (StrAlg.CanRun) THEN
  					StrAlg.isRuning := TRUE;
  					StrAlg.isEnded := FALSE;
  					StrAlg.hasError := FALSE;
  					(*****************       OnRun       *****************)

                                                    algManager.nMode:=ModeGpa.MODE_PUSKV;
                                                    resetAndDisable(alg:=algoritms.ppu);
                                                    algoritms.puskOilSystem.inCanRun:= TRUE;
                                                    algoritms.engineRun.inCanRun:= TRUE;
                                                    runPhase(puskOilSystem);

  					cmd_for_Status := cmd;
  					source_for_Status := source;
  					command_error_for_Status := 0;
  				ELSE
  					StrAlg.isRuning := FALSE;
  					StrAlg.isEnded := FALSE;
  					StrAlg.hasError 	:= FALSE;

  					cmd_for_Status := 0;
  					source_for_Status := source;
  					command_error_for_Status := cmd;
  				END_IF;
  		(*cmdReset*) 2: 	StrAlg.isRuning := FALSE;
  				StrAlg.isEnded := FALSE;
  				StrAlg.hasError 	:= FALSE;

                                           (*****************       OnReset       *****************)
                                          waitReset(IN:=FALSE);
                                          _resetQuestion1:=FALSE;
                                          _resetQuestion2:=FALSE;
                                          resetPhase(puskOilSystem);
                                          resetPhase(runningEngine);
                                          resetPhase(mvOff);
                                          resetPhase(pnsOn);
                                          resetPhase(wait600);
                                          resetPhase(AutoNUoff);
                                          resetPhase(nu1Off);
                                          resetPhase(nu2Off);
                                          resetPhase(pnsWaitOff);
  	                              resetPhase(autoAvomOff);
                                          resetPhase(Avom1Off);
                                          resetPhase(Avom2Off);
                                          resetPhase(testUnsuccessful);

                                          resetQuestion(questionEngine);
                                          resetQuestion(questionMVoff);

                                          StrAlg.inOpcCommandsDisabled:=FALSE;

  				cmd_for_Status := cmd;
  				source_for_Status := source;
  				command_error_for_Status := 0;
  	END_CASE;
  	resetCmdTimer(IN := false);
  	resetCmdTimerPriznak := TRUE;
  END_IF;
  lastCmd := cmd;

  resetCmdTimer(IN := resetCmdTimerPriznak, PT := T#5S);
  IF resetCmdTimer.Q THEN
  	resetCmdTimerPriznak := FALSE;
  	source_for_Status := 0;
  	cmd_for_Status := 0;
  	command_error_for_Status := 0;
  END_IF;

  StrAlg.Start:= puskOilSystem.startStatus
              OR runningEngine.startStatus
              OR mvOff.startStatus
              OR pnsOn.startStatus
              OR wait600.startStatus
              OR AutoNUoff.startStatus
              OR nu1Off.startStatus
              OR nu2Off.startStatus
              OR pnsWaitOff.startStatus
              OR testUnsuccessful.startStatus;

  StrAlg.Error:=  puskOilSystem.errorStatus
              OR runningEngine.errorStatus
              OR mvOff.errorStatus
              OR pnsOn.errorStatus
              OR wait600.errorStatus
              OR AutoNUoff.errorStatus
              OR nu1Off.errorStatus
              OR nu2Off.errorStatus
              OR pnsWaitOff.errorStatus
              OR testUnsuccessful.errorStatus;

  StrAlg.Top:=   puskOilSystem.topStatus
              OR runningEngine.topStatus
              OR mvOff.topStatus
              OR pnsOn.topStatus
              OR wait600.topStatus
              OR AutoNUoff.topStatus
              OR nu1Off.topStatus
              OR nu2Off.topStatus
              OR pnsWaitOff.topStatus
              OR testUnsuccessful.topStatus;

  (*TODO: TYPE PROGRAM CODE HERE*)
  StrAlg.status :=  SHL(BYTE_TO_DWORD(source_for_Status), 29)
  			OR SHL(BYTE_TO_DWORD(cmd_for_Status), 26)
  			OR SHL(BYTE_TO_DWORD(command_error_for_Status), 23)
  			OR SHL(BOOL_TO_DWORD(StrAlg.OpcCommandsDisabled ), 21)
  			OR SHL(BOOL_TO_DWORD(StrAlg.hasError),4)
  			OR SHL(BOOL_TO_DWORD(StrAlg.CanRun),2)
  			OR SHL(BOOL_TO_DWORD(StrAlg.isEnded),1)
  			OR BOOL_TO_DWORD(StrAlg.isRuning);
END_FUNCTION_BLOCK

FUNCTION_BLOCK testdPmgAlg
  VAR_IN_OUT
    StrAlg : struct_Alg;
  END_VAR
  VAR
    puskOilSystem : struct_PhaseAlgoritm;
  END_VAR
  VAR_IN_OUT
    algContinue : struct_Question;
  END_VAR
  VAR
    nuOff : struct_PhaseAlgoritm;
    dPmgAi : struct_PhaseAlgoritm;
    dPmgDi : struct_PhaseAlgoritm;
    nuOn : struct_PhaseAlgoritm;
    noRezrv : struct_PhaseAlgoritm;
    BreakTest : struct_PhaseAlgoritm;
    testUnsuccessful : struct_PhaseAlgoritm;
    pnsOff : struct_PhaseAlgoritm;
    stopANU : struct_PhaseAlgoritm;
    Ust_dPLow : struct_PhaseAlgoritm;
    nu1Off : struct_PhaseAlgoritm;
    nu2Off : struct_PhaseAlgoritm;
    stopNU1 : struct_PhaseAlgoritm;
    stopNU2 : struct_PhaseAlgoritm;
    fb_puskOilSystem : fb_ph_algoritm;
    fb_algContinue : fb_Question;
    fb_nuOff : fb_ph_CustomPhase;
    fb_dPmgAi : fb_ph_WaitAnalogValue;
    fb_dPmgDi : fb_ph_CustomPhase;
    fb_nuOn : fb_ph_CustomPhase;
    fb_noRezrv : fb_ph_CustomPhase;
    fb_BreakTest : fb_ph_Timer;
    fb_testUnsuccessful : fb_ph_CustomPhase;
    fb_pnsOff : fb_ph_Switch;
    fb_stopANU : fb_ph_CustomPhase;
    fb_nu1Off : fb_ph_OilPump;
    fb_nu2Off : fb_ph_OilPump;
    fb_stopNU1 : fb_ph_OilPump;
    fb_stopNU2 : fb_ph_OilPump;
    _sunpackerCommand : fb_sunpackerCommand;
    _DualStateImAction : TYPE_DualStateImAction;
    _Answers : TYPE_Answers;
    _statusDualInput : TYPE_statusDualInput;
    _StatusAi : TYPE_StatusAi;
    _PhaseAlgoritmAction : TYPE_PhaseAlgoritmAction;
    source : BYTE;
    cmd : BYTE;
    lastCmd : BYTE;
    source_for_Status : BYTE;
    cmd_for_Status : BYTE;
    command_error_for_Status : BYTE;
    resetCmdTimer : TON;
    resetCmdTimerPriznak : BOOL;
    onInit : BOOL;
    _resetQuestion : BOOL;
    waitReset : TON;
    WaitOnNU : TON;
  END_VAR
  VAR_EXTERNAL
    IM : ImConfig;
    algoritms : AlgoritmsConfig;
    ai : AiConfig;
    AlgTimers : struct_AlgTimers;
    ModeGpa : TYPE_ModeGpa;
    algManager : struct_AlgoritmsManager;
    protections : ProtectionsConfig;
    NotHasRezervNU : BOOL;
  END_VAR

  IF NOT onInit THEN

      fb_puskOilSystem(phaseNumber:=0, act:=_run, waitCompletion:=TRUE);
          algContinue.AnswerVariants:=_Answers.ANS_YES;
              fb_nuOff(phaseNumber:=1);
             fb_dPmgAi(phaseNumber:=2);
             fb_dPmgDi(phaseNumber:=3);
               fb_nuOn(phaseNumber:=4);
            fb_noRezrv(phaseNumber:=5);
   fb_testUnsuccessful(phaseNumber:=6);
          fb_BreakTest(phaseNumber:=7, delay:=T#10S);
             fb_pnsOff(phaseNumber:=8, act:=_off);
            fb_stopANU(phaseNumber:=9);
             fb_nu1Off(phaseNumber:=11, act:=_off);
             fb_nu2Off(phaseNumber:=12, act:=_off);
            fb_stopNU1(phaseNumber:=15, act:=_off);
            fb_stopNU2(phaseNumber:=16, act:=_off);
  onInit:=TRUE;
  END_IF;

      fb_puskOilSystem(StrPh:=puskOilSystem, alg:=algoritms.puskOilSystem);
        fb_algContinue(StrQ:=algContinue);
              fb_nuOff(StrPh:=nuOff);
             (*fb_dPmgAi(StrPh:=dPmgAi, ai:=ai.Tmasla_MB, less:=im.testdPmg_Ust_dPLow.Value);*)
             fb_dPmgDi(StrPh:=dPmgDi);
               fb_nuOn(StrPh:=nuOn);
            fb_noRezrv(StrPh:=noRezrv);
   fb_testUnsuccessful(StrPh:=testUnsuccessful);
          fb_BreakTest(StrPh:=BreakTest, timer:=AlgTimers.testdPmg_BreakTest);
             fb_pnsOff(StrPh:=pnsOff, Im:=Im.pns);
            fb_stopANU(StrPh:=stopANU);
             fb_nu1Off(StrPh:=nu1Off, Im:=Im.nu1);
             fb_nu2Off(StrPh:=nu2Off, Im:=Im.nu2);
            fb_stopNU1(StrPh:=stopNU1, Im:=Im.nu1);
            fb_stopNU2(StrPh:=stopNU2, Im:=Im.nu2);

  StrAlg.CanRun := StrAlg.inCanRun;
  StrAlg.OpcCommandsDisabled := StrAlg.inOpcCommandsDisabled;

  IF StrAlg.isRuning THEN

      StrAlg.hasError := pnsOff.error OR nu1Off.error OR nu2Off.error
      OR stopNU1.error OR stopNU2.error OR testUnsuccessful.error;

      IF puskOilSystem.top THEN
           IF NOT _resetQuestion THEN
           askQuestion(algContinue);
            _resetQuestion:=TRUE;
           END_IF;
      END_IF;

      IF algContinue.answer = _Answers.ANS_YES AND NOT nuOff.top THEN

          runPhase(nuOff);

          IF Im.nu1.onStatus = _statusDualInput.STATUS_ON THEN
  		runPhase(nu1Off);
          END_IF;

          IF Im.nu2.onStatus = _statusDualInput.STATUS_ON THEN
  		runPhase(nu2Off);
          END_IF;

          resetQuestion(algContinue);

      END_IF;

      IF nuOff.start AND NOT nuOff.top THEN
            runPhase(BreakTest);
  	nuOff.top:= Im.nu1.onStatus = _statusDualInput.STATUS_Off
                    AND Im.nu2.onStatus = _statusDualInput.STATUS_Off;
      END_IF;

      IF nuOff.top THEN

          runPhase(dPmgAi);
          runPhase(dPmgDi);
      END_IF;

      (*IF dPmgDi.start AND NOT dPmgDi.top THEN
          dPmgDi.top:=Im.SingleSignals.dP_oilgaz_low.q;
      END_IF;*)

      IF dPmgAi.top AND dPmgDi.top THEN
          runPhase(nuOn);
          runPhase(noRezrv);
      END_IF;

      IF noRezrv.start AND NOT noRezrv.top THEN
          noRezrv.top:=NotHasRezervNU;
      END_IF;

       IF nuOn.start AND (NOT WaitOnNU.Q) THEN
          WaitOnNU(IN:=Im.nu1.onStatus = _statusDualInput.STATUS_On OR
              Im.nu2.onStatus = _statusDualInput.STATUS_On, PT:=T#2S);
          nuOn.top:=Im.nu1.onStatus = _statusDualInput.STATUS_On OR
              Im.nu2.onStatus = _statusDualInput.STATUS_On;
      END_IF;

      IF  WaitOnNU.Q AND noRezrv.top THEN
          ai.Tmasla_MB.Disabled_LA:=TRUE;
          ai.Tmasla_MB.Disabled_LW:=TRUE;
          (*IM.SingleSignals.dP_oilgaz_low.Disabled_Sig:=TRUE;
          IM.SingleSignals.P_oil_low.Disabled_Sig:=TRUE;*)
          ai.Pmasla_posle_GNS.Disabled_LA:=TRUE;
          ai.Pmasla_posle_GNS.Disabled_LW:=TRUE;
          ai.Pmasla_posle_NU.Disabled_LW:=TRUE;

          resetAiProtection(protections.Os_sdvig_nagnetatelja_minus);
          (*resetDiProtection(protections.Vibro_skorost_OP_shesterni_RED_T6);*)
          resetAiProtection(protections.Os_sdvig_nagnetatelja_plus);
          (*resetDiProtection(protections.Vibro_skorost_OP_shesterni_RED_T5);*)

          resetIfRunning(algoritms.autoNu);
          resetIfRunning(algoritms.AutoPns);

          runPhase(stopANU);
          runPhase(pnsOff);

          runPhase(stopNU1);
          runPhase(stopNU2);

      END_IF;

      IF stopANU.start AND NOT stopANU.top THEN

  	stopANU.top:= Im.nu1.onStatus = _statusDualInput.STATUS_Off AND
                          Im.nu2.onStatus = _statusDualInput.STATUS_Off;
      END_IF;

      IF BreakTest.top AND NOT pnsOff.top THEN
  	testUnsuccessful.error:=TRUE;
      END_IF;

      IF pnsOff.top AND stopANU.top THEN
            resetPhase(BreakTest);
  	waitReset(IN:=TRUE, PT:= T#3S);
      END_IF;

      IF waitReset.Q THEN
          algManager.nMode:=ModeGpa.MODE_STOP;
          resetIfRunning(StrAlg);
      END_IF;

      StrAlg.isEnded:= pnsOff.top AND stopANU.top;

  END_IF;

  StrAlg.CanRun := StrAlg.inCanRun;
  StrAlg.OpcCommandsDisabled := StrAlg.inOpcCommandsDisabled;

  (* ---- Если управление с ВУ заблокировано, то  передаем команду из алгоритма ---- *)
  IF StrAlg.inOpcCommandsDisabled THEN
  	StrAlg.inCommand := StrAlg.inCommand_Alg;
  ELSE (* иначе передаем команду с АРМа*)
  	StrAlg.inCommand := StrAlg.inCommand_ARM;
  END_IF;

  _sunpackerCommand(command := StrAlg.inCommand);
  	source := _sunpackerCommand.source;
  	cmd := _sunpackerCommand.cmd;

  IF cmd <> 0 AND lastCmd <> cmd AND (((NOT StrAlg.opcCommandsDisabled) AND source > 0) OR source = 0) then
  	CASE BYTE_TO_INT(cmd) OF
  		(*cmdRun*) 1: 	IF (StrAlg.CanRun) THEN
  					StrAlg.isRuning := TRUE;
  					StrAlg.isEnded := FALSE;
  					StrAlg.hasError := FALSE;
  					(*****************       OnRun       *****************)

                                                    algManager.nMode:=ModeGpa.MODE_TESTDPMG;
                                                    resetAndDisable(alg:=algoritms.ppu);
                                                    algoritms.puskOilSystem.inCanRun:= TRUE;
                                                    runPhase(puskOilSystem);

  					cmd_for_Status := cmd;
  					source_for_Status := source;
  					command_error_for_Status := 0;
  				ELSE
  					StrAlg.isRuning := FALSE;
  					StrAlg.isEnded := FALSE;
  					StrAlg.hasError 	:= FALSE;

  					cmd_for_Status := 0;
  					source_for_Status := source;
  					command_error_for_Status := cmd;
  				END_IF;
  		(*cmdReset*) 2: 	StrAlg.isRuning := FALSE;
  				StrAlg.isEnded := FALSE;
  				StrAlg.hasError 	:= FALSE;

                                           (*****************       OnReset       *****************)
                                          waitReset(IN:=FALSE);
                                          WaitOnNU(IN:=FALSE);
                                          _resetQuestion:=FALSE;
                                          ai.Pmasla_posle_GNS.Disabled_LA:=TRUE;
                                          ai.Pmasla_posle_GNS.Disabled_LW:=TRUE;
                                          ai.Pmasla_posle_NU.Disabled_LW:=TRUE;
                                          (*IM.SingleSignals.P_oil_low.Disabled_Sig:=TRUE;
                                          IM.SingleSignals.dP_oilgaz_low.Disabled_Sig:=TRUE;*)
                                          ai.Tmasla_MB.Disabled_LA:=TRUE;
                                          ai.Tmasla_MB.Disabled_LW:=TRUE;
                                          resetAiProtection(protections.Os_sdvig_nagnetatelja_minus);
                                          (*resetDiProtection(protections.Vibro_skorost_OP_shesterni_RED_T6);*)
                                          resetAiProtection(protections.Os_sdvig_nagnetatelja_plus);
                                          (*resetDiProtection(protections.Vibro_skorost_OP_shesterni_RED_T5);*)

                                          resetPhase(puskOilSystem);
                                          resetPhase(nuOff);
                                          resetPhase(dPmgAi);
                                          resetPhase(dPmgDi);
                                          resetPhase(nuOn);
                                          resetPhase(noRezrv);
                                          resetPhase(BreakTest);
                                          resetPhase(testUnsuccessful);
                                          resetPhase(pnsOff);
                                          resetPhase(stopANU);
                                          resetPhase(nu1Off);
                                          resetPhase(nu2Off);
                                          resetPhase(stopNU1);
                                          resetPhase(stopNU2);

                                          resetQuestion(algContinue);

                                          StrAlg.inOpcCommandsDisabled:=FALSE;

  				cmd_for_Status := cmd;
  				source_for_Status := source;
  				command_error_for_Status := 0;
  	END_CASE;
  	resetCmdTimer(IN := false);
  	resetCmdTimerPriznak := TRUE;
  END_IF;
  lastCmd := cmd;

  resetCmdTimer(IN := resetCmdTimerPriznak, PT := T#5S);
  IF resetCmdTimer.Q THEN
  	resetCmdTimerPriznak := FALSE;
  	source_for_Status := 0;
  	cmd_for_Status := 0;
  	command_error_for_Status := 0;
  END_IF;

  StrAlg.Start:= puskOilSystem.startStatus
              OR nuOff.startStatus
              OR dPmgAi.startStatus
              OR dPmgDi.startStatus
              OR nuOn.startStatus
              OR noRezrv.startStatus
              OR BreakTest.startStatus
              OR testUnsuccessful.startStatus
              OR pnsOff.startStatus
              OR stopANU.startStatus
              OR nu1Off.startStatus
              OR nu2Off.startStatus;

  StrAlg.Error:=  puskOilSystem.errorStatus
              OR nuOff.errorStatus
              OR dPmgAi.errorStatus
              OR dPmgDi.errorStatus
              OR nuOn.errorStatus
              OR noRezrv.errorStatus
              OR BreakTest.errorStatus
              OR testUnsuccessful.errorStatus
              OR pnsOff.errorStatus
              OR stopANU.errorStatus
              OR nu1Off.errorStatus
              OR nu2Off.errorStatus;

  StrAlg.Top:=   puskOilSystem.topStatus
              OR nuOff.topStatus
              OR dPmgAi.topStatus
              OR dPmgDi.topStatus
              OR nuOn.topStatus
              OR noRezrv.topStatus
              OR BreakTest.topStatus
              OR testUnsuccessful.topStatus
              OR pnsOff.topStatus
              OR stopANU.topStatus
              OR nu1Off.topStatus
              OR nu2Off.topStatus;

  (*TODO: TYPE PROGRAM CODE HERE*)
  StrAlg.status :=  SHL(BYTE_TO_DWORD(source_for_Status), 29)
  			OR SHL(BYTE_TO_DWORD(cmd_for_Status), 26)
  			OR SHL(BYTE_TO_DWORD(command_error_for_Status), 23)
  			OR SHL(BOOL_TO_DWORD(StrAlg.OpcCommandsDisabled ), 21)
  			OR SHL(BOOL_TO_DWORD(StrAlg.hasError),4)
  			OR SHL(BOOL_TO_DWORD(StrAlg.CanRun),2)
  			OR SHL(BOOL_TO_DWORD(StrAlg.isEnded),1)
  			OR BOOL_TO_DWORD(StrAlg.isRuning);
END_FUNCTION_BLOCK

FUNCTION_BLOCK fb_ph_AIprotection
  VAR_IN_OUT
    StrAiP : struct_AiProtection;
  END_VAR
  VAR_INPUT
    act : TYPE_PhaseAlgoritmAction;
    PhaseNumber : UINT;
  END_VAR
  VAR_IN_OUT
    StrPh : struct_PhaseAlgoritm;
  END_VAR
  VAR
    CommandFault_Trig : R_TRIG;
    reset_Trig : R_TRIG;
    _statusDualInput : TYPE_statusDualInput;
  END_VAR

  IF StrPh.run AND NOT StrPh.start THEN
  	StrPh.start := TRUE;
  	StrPh.top := FALSE;
  	StrPh.error := FALSE;
            StrPh.run:=FALSE;

  	CASE act OF
  		(*PhaseAlgoritmAction.run*)    _run : runAiProtection(StrAiP); (*cmd_run*)
  		(*PhaseAlgoritmAction.reset*)_reset : resetAiProtection(StrAiP); (*cmd_reset*)
  	END_CASE;
  END_IF;

  IF StrPh.start AND NOT StrPh.top THEN
                      CommandFault_Trig(CLK := StrAiP.hasError);
                      IF CommandFault_Trig.Q THEN
  	          StrPh.error := TRUE;
                      END_IF;

  		CASE act OF
  		(*PhaseAlgoritmAction.run*)    _run:    StrPh.top:=StrAiP.isRunning;

  		(*PhaseAlgoritmAction.reset*) _reset:   StrPh.top := NOT StrAiP.isRunning;
  		END_CASE;

  END_IF;

  IF StrPh.top THEN
  StrPh.error := FALSE;
  END_IF;

  reset_Trig(CLK := StrPh.reset);
  IF reset_Trig.Q THEN
            StrPh.start := FALSE;
  	StrPh.error := FALSE;
  	StrPh.top := FALSE;
            StrPh.run:=FALSE;
            StrPh.reset:=FALSE;
  END_IF;

  StrPh.startStatus := SHL(BOOL_TO_DWORD(StrPh.start), PhaseNumber);
  StrPh.errorStatus := SHL(BOOL_TO_DWORD(StrPh.error), PhaseNumber);
  StrPh.topStatus := SHL(BOOL_TO_DWORD(StrPh.top), PhaseNumber);
END_FUNCTION_BLOCK

FUNCTION_BLOCK testPmsAlg
  VAR_IN_OUT
    StrAlg : struct_Alg;
    algContinue : struct_Question;
  END_VAR
  VAR
    pnsOn : struct_PhaseAlgoritm;
    PmsUp : struct_PhaseAlgoritm;
    runProtecrionAi : struct_PhaseAlgoritm;
    pnsOff : struct_PhaseAlgoritm;
    BreakTest : struct_PhaseAlgoritm;
    LowOilPS : struct_PhaseAlgoritm;
    LowOilAS : struct_PhaseAlgoritm;
    testUnsuccessful : struct_PhaseAlgoritm;
    fb_pnsOn : fb_ph_Switch;
    fb_PmsUp : fb_ph_WaitAnalogValue;
    fb_algContinue : fb_Question;
    fb_runProtecrionAi : fb_ph_AIprotection;
    fb_pnsOff : fb_ph_Switch;
    fb_BreakTest : fb_ph_Timer;
    fb_LowOilPS : fb_ph_CustomPhase;
    fb_LowOilAS : fb_ph_CustomPhase;
    fb_testUnsuccessful : fb_ph_CustomPhase;
    _sunpackerCommand : fb_sunpackerCommand;
    _DualStateImAction : TYPE_DualStateImAction;
    _Answers : TYPE_Answers;
    _statusDualInput : TYPE_statusDualInput;
    _StatusAi : TYPE_StatusAi;
    _PhaseAlgoritmAction : TYPE_PhaseAlgoritmAction;
    source : BYTE;
    cmd : BYTE;
    lastCmd : BYTE;
    source_for_Status : BYTE;
    cmd_for_Status : BYTE;
    command_error_for_Status : BYTE;
    resetCmdTimer : TON;
    resetCmdTimerPriznak : BOOL;
    onInit : BOOL;
    _resetQuestion : BOOL;
    waitReset : TON;
  END_VAR
  VAR_EXTERNAL
    IM : ImConfig;
    algoritms : AlgoritmsConfig;
    ai : AiConfig;
    AlgTimers : struct_AlgTimers;
    ModeGpa : TYPE_ModeGpa;
    algManager : struct_AlgoritmsManager;
    protections : ProtectionsConfig;
  END_VAR

  IF NOT onInit THEN

                     fb_pnsOn(phaseNumber:=0, act:=_on);
          algContinue.AnswerVariants:=_Answers.ANS_YES;
                     fb_PmsUp(phaseNumber:=1);
           fb_runProtecrionAi(phaseNumber:=3, act:=_run);
                    fb_pnsOff(phaseNumber:=4, act:=_off);
                 fb_BreakTest(phaseNumber:=5, delay:=T#120S);
                  fb_LowOilPS(phaseNumber:=6);
                  fb_LowOilAS(phaseNumber:=7);
          fb_testUnsuccessful(phaseNumber:=8);

  onInit:=TRUE;
  END_IF;

              fb_pnsOn(StrPh:=pnsOn, Im:=IM.pns);
        fb_algContinue(StrQ:=algContinue);
              fb_PmsUp(StrPh:=PmsUp, ai:=ai.Pmasla_posle_GNS, more:=ai.Pmasla_posle_GNS.LW);
    fb_runProtecrionAi(StrPh:=runProtecrionAi, StrAiP:=protections.Os_sdvig_nagnetatelja_minus);
             fb_pnsOff(StrPh:=pnsOff, Im:=IM.pns);
          fb_BreakTest(StrPh:=BreakTest, timer:=AlgTimers.testPms_BreakTest);
           fb_LowOilPS(StrPh:=LowOilPS);
           fb_LowOilAS(StrPh:=LowOilAS);
   fb_testUnsuccessful(StrPh:=testUnsuccessful);

  StrAlg.CanRun := StrAlg.inCanRun;
  StrAlg.OpcCommandsDisabled := StrAlg.inOpcCommandsDisabled;

  IF StrAlg.isRuning THEN

      StrAlg.hasError := pnsOn.error OR pnsOff.error OR testUnsuccessful.error;

      IF pnsOn.top THEN
           runPhase(PmsUp);
      END_IF;

      IF PmsUp.top THEN
           runPhase(runProtecrionAi);
      END_IF;

      IF runProtecrionAi.top THEN
           (*IM.SingleSignals.P_oil_low.Disabled_Sig:=FALSE;*)
           ai.Pmasla_posle_GNS.Disabled_LA:=FALSE;
           ai.Pmasla_posle_GNS.Disabled_LW:=FALSE;
           ai.Pmasla_posle_NU.Disabled_LW:=FALSE;
               IF NOT _resetQuestion THEN
                   askQuestion(algContinue);
                   _resetQuestion:=TRUE;
               END_IF;
      END_IF;

      IF algContinue.answer = _Answers.ANS_YES THEN

          runPhase(BreakTest);
          runPhase(pnsOff);
          runPhase(LowOilPS);
          runPhase(LowOilAS);
          resetQuestion(algContinue);

      END_IF;

      IF 	LowOilPS.start AND NOT LowOilPS.top THEN
  	LowOilPS.top:= ai.Pmasla_posle_GNS.interval = _statusAi.LW;
      END_IF;
      IF 	LowOilAS.start AND NOT LowOilAS.top THEN
  	LowOilAS.top:= ai.Pmasla_posle_GNS.interval = _statusAi.LA;
      END_IF;

      IF LowOilPS.top AND LowOilAS.top THEN
            resetPhase(BreakTest);
            waitReset(IN:=TRUE, PT:= T#3S);
      END_IF;

      IF BreakTest.top AND StrAlg.isEnded THEN
  	testUnsuccessful.error:=TRUE;
      END_IF;

      IF waitReset.Q THEN
          algManager.nMode:=ModeGpa.MODE_STOP;
          resetIfRunning(StrAlg);
      END_IF;

      StrAlg.isEnded:= LowOilPS.top AND LowOilAS.top;

  END_IF;

  StrAlg.CanRun := StrAlg.inCanRun;
  StrAlg.OpcCommandsDisabled := StrAlg.inOpcCommandsDisabled;

  (* ---- Если управление с ВУ заблокировано, то  передаем команду из алгоритма ---- *)
  IF StrAlg.inOpcCommandsDisabled THEN
  	StrAlg.inCommand := StrAlg.inCommand_Alg;
  ELSE (* иначе передаем команду с АРМа*)
  	StrAlg.inCommand := StrAlg.inCommand_ARM;
  END_IF;

  _sunpackerCommand(command := StrAlg.inCommand);
  	source := _sunpackerCommand.source;
  	cmd := _sunpackerCommand.cmd;

  IF cmd <> 0 AND lastCmd <> cmd AND (((NOT StrAlg.opcCommandsDisabled) AND source > 0) OR source = 0) then
  	CASE BYTE_TO_INT(cmd) OF
  		(*cmdRun*) 1: 	IF (StrAlg.CanRun) THEN
  					StrAlg.isRuning := TRUE;
  					StrAlg.isEnded := FALSE;
  					StrAlg.hasError := FALSE;
  					(*****************       OnRun       *****************)

                                                    algManager.nMode:=ModeGpa.MODE_TESTPMS;
                                                    resetAndDisable(alg:=algoritms.ppu);
                                                    runPhase(pnsOn);

  					cmd_for_Status := cmd;
  					source_for_Status := source;
  					command_error_for_Status := 0;
  				ELSE
  					StrAlg.isRuning := FALSE;
  					StrAlg.isEnded := FALSE;
  					StrAlg.hasError 	:= FALSE;

  					cmd_for_Status := 0;
  					source_for_Status := source;
  					command_error_for_Status := cmd;
  				END_IF;
  		(*cmdReset*) 2: 	StrAlg.isRuning := FALSE;
  				StrAlg.isEnded := FALSE;
  				StrAlg.hasError 	:= FALSE;

                                           (*****************       OnReset       *****************)
                                          waitReset(IN:=FALSE);
                                          _resetQuestion:=FALSE;
                                          ai.Pmasla_posle_GNS.Disabled_LA:=TRUE;
                                          ai.Pmasla_posle_GNS.Disabled_LW:=TRUE;
                                          ai.Pmasla_posle_NU.Disabled_LW:=TRUE;
                                         (* IM.SingleSignals.P_oil_low.Disabled_Sig:=TRUE;*)
                                          resetAiProtection(protections.Os_sdvig_nagnetatelja_minus);

                                          resetPhase(pnsOn);
                                          resetPhase(PmsUp);
                                          resetPhase(runProtecrionAi);
                                          resetPhase(pnsOff);
                                          resetPhase(BreakTest);
                                          resetPhase(LowOilPS);
                                          resetPhase(LowOilAS);
                                          resetPhase(testUnsuccessful);

                                          resetQuestion(algContinue);

                                          StrAlg.inOpcCommandsDisabled:=FALSE;

  				cmd_for_Status := cmd;
  				source_for_Status := source;
  				command_error_for_Status := 0;
  	END_CASE;
  	resetCmdTimer(IN := false);
  	resetCmdTimerPriznak := TRUE;
  END_IF;
  lastCmd := cmd;

  resetCmdTimer(IN := resetCmdTimerPriznak, PT := T#5S);
  IF resetCmdTimer.Q THEN
  	resetCmdTimerPriznak := FALSE;
  	source_for_Status := 0;
  	cmd_for_Status := 0;
  	command_error_for_Status := 0;
  END_IF;

  StrAlg.Start:= pnsOn.startStatus
              OR PmsUp.startStatus
              OR runProtecrionAi.startStatus
              OR pnsOff.startStatus
              OR BreakTest.startStatus
              OR LowOilPS.startStatus
              OR LowOilAS.startStatus
              OR testUnsuccessful.startStatus;

  StrAlg.Error:= pnsOn.errorStatus
              OR PmsUp.errorStatus
              OR runProtecrionAi.errorStatus
              OR pnsOff.errorStatus
              OR BreakTest.errorStatus
              OR LowOilPS.errorStatus
              OR LowOilAS.errorStatus
              OR testUnsuccessful.errorStatus;

  StrAlg.Top:=   pnsOn.topStatus
              OR PmsUp.topStatus
              OR runProtecrionAi.topStatus
              OR pnsOff.topStatus
              OR BreakTest.topStatus
              OR LowOilPS.topStatus
              OR LowOilAS.topStatus
              OR testUnsuccessful.topStatus;

  (*TODO: TYPE PROGRAM CODE HERE*)
  StrAlg.status :=  SHL(BYTE_TO_DWORD(source_for_Status), 29)
  			OR SHL(BYTE_TO_DWORD(cmd_for_Status), 26)
  			OR SHL(BYTE_TO_DWORD(command_error_for_Status), 23)
  			OR SHL(BOOL_TO_DWORD(StrAlg.OpcCommandsDisabled ), 21)
  			OR SHL(BOOL_TO_DWORD(StrAlg.hasError),4)
  			OR SHL(BOOL_TO_DWORD(StrAlg.CanRun),2)
  			OR SHL(BOOL_TO_DWORD(StrAlg.isEnded),1)
  			OR BOOL_TO_DWORD(StrAlg.isRuning);
END_FUNCTION_BLOCK

FUNCTION_BLOCK ApuskAlg
  VAR_IN_OUT
    StrAlg : struct_Alg;
  END_VAR
  VAR
    runOilsystem : struct_PhaseAlgoritm;
    runEngine : struct_PhaseAlgoritm;
    filling : struct_PhaseAlgoritm;
    fb_runOilsystem : fb_ph_algoritm;
    fb_runEngine : fb_ph_algoritm;
    fb_filling : fb_ph_algoritm;
    _sunpackerCommand : fb_sunpackerCommand;
    _PhaseAlgoritmAction : TYPE_PhaseAlgoritmAction;
    _statusDualInput : TYPE_statusDualInput;
    source : BYTE;
    cmd : BYTE;
    lastCmd : BYTE;
    source_for_Status : BYTE;
    cmd_for_Status : BYTE;
    command_error_for_Status : BYTE;
    resetCmdTimer : TON;
    resetCmdTimerPriznak : BOOL;
    onInit : BOOL;
    waitReset : TON;
  END_VAR
  VAR_EXTERNAL
    algoritms : AlgoritmsConfig;
    ModeGpa : TYPE_ModeGpa;
    algManager : struct_AlgoritmsManager;
    IM : ImConfig;
  END_VAR

  IF NOT onInit THEN

           fb_runOilsystem(phaseNumber:=0, act:=_run, waitCompletion:=TRUE);
              fb_runEngine(phaseNumber:=1, act:=_run, waitCompletion:=TRUE);
                fb_filling(phaseNumber:=2, act:=_run, waitCompletion:=TRUE);

  onInit:=TRUE;
  END_IF;

           fb_runOilsystem(StrPh:=runOilsystem, alg:=algoritms.puskOilSystem);
              fb_runEngine(StrPh:=runEngine, alg:=algoritms.engineRun);
                fb_filling(StrPh:=filling, alg:=algoritms.filling);

  StrAlg.CanRun := StrAlg.inCanRun;
  StrAlg.OpcCommandsDisabled := StrAlg.inOpcCommandsDisabled;

  IF StrAlg.isRuning THEN

      StrAlg.hasError := runOilsystem.error OR runEngine.error OR filling.error;

      IF runOilsystem.top THEN
           runPhase(runEngine);
      END_IF;

      IF runEngine.top THEN
           runPhase(filling);
      END_IF;

      IF filling.top THEN
            waitReset(IN:=TRUE, PT:= T#2S);
      END_IF;

      IF waitReset.Q THEN

          IF Im.kran6.onStatus = _statusDualInput.STATUS_On THEN
  	algManager.nMode:= ModeGpa.MODE_WORK_Ring;
          END_IF;
          IF Im.kran6.onStatus = _statusDualInput.STATUS_Off THEN
  	algManager.nMode:= ModeGpa.MODE_WORK_Line;
          END_IF;

          resetIfRunning(StrAlg);
      END_IF;

      StrAlg.isEnded:= filling.top;

  END_IF;

  StrAlg.CanRun := StrAlg.inCanRun;
  StrAlg.OpcCommandsDisabled := StrAlg.inOpcCommandsDisabled;

  (* ---- Если управление с ВУ заблокировано, то  передаем команду из алгоритма ---- *)
  IF StrAlg.inOpcCommandsDisabled THEN
  	StrAlg.inCommand := StrAlg.inCommand_Alg;
  ELSE (* иначе передаем команду с АРМа*)
  	StrAlg.inCommand := StrAlg.inCommand_ARM;
  END_IF;

  _sunpackerCommand(command := StrAlg.inCommand);
  	source := _sunpackerCommand.source;
  	cmd := _sunpackerCommand.cmd;

  IF cmd <> 0 AND lastCmd <> cmd AND (((NOT StrAlg.opcCommandsDisabled) AND source > 0) OR source = 0) then
  	CASE BYTE_TO_INT(cmd) OF
  		(*cmdRun*) 1: 	IF (StrAlg.CanRun) THEN
  					StrAlg.isRuning := TRUE;
  					StrAlg.isEnded := FALSE;
  					StrAlg.hasError := FALSE;
  					(*****************       OnRun       *****************)

                                                    algoritms.puskOilSystem.inCanRun:= TRUE	;
                                                    algoritms.filling.inCanRun:= TRUE	;
                                                    algoritms.engineRun.inCanRun:= TRUE	;

                                                    algManager.nMode:=ModeGpa.MODE_APUSK;
                                                    (*impulseSO(Im.SingleOutputs.VzvodBREO);*)
                                                    runPhase(runOilsystem);

  					cmd_for_Status := cmd;
  					source_for_Status := source;
  					command_error_for_Status := 0;
  				ELSE
  					StrAlg.isRuning := FALSE;
  					StrAlg.isEnded := FALSE;
  					StrAlg.hasError 	:= FALSE;

  					cmd_for_Status := 0;
  					source_for_Status := source;
  					command_error_for_Status := cmd;
  				END_IF;
  		(*cmdReset*) 2: 	StrAlg.isRuning := FALSE;
  				StrAlg.isEnded := FALSE;
  				StrAlg.hasError 	:= FALSE;

                                           (*****************       OnReset       *****************)
                                          waitReset(IN:=FALSE);
                                          StrAlg.inCanRun:=FALSE;

                                          resetPhase(runOilsystem);
                                          resetPhase(runEngine);
                                          resetPhase(filling);

                                          StrAlg.inOpcCommandsDisabled:=FALSE;

  				cmd_for_Status := cmd;
  				source_for_Status := source;
  				command_error_for_Status := 0;
  	END_CASE;
  	resetCmdTimer(IN := false);
  	resetCmdTimerPriznak := TRUE;
  END_IF;
  lastCmd := cmd;

  resetCmdTimer(IN := resetCmdTimerPriznak, PT := T#5S);
  IF resetCmdTimer.Q THEN
  	resetCmdTimerPriznak := FALSE;
  	source_for_Status := 0;
  	cmd_for_Status := 0;
  	command_error_for_Status := 0;
  END_IF;

  StrAlg.Start:= runOilsystem.startStatus
              OR runEngine.startStatus
              OR filling.startStatus;

  StrAlg.Error:= runOilsystem.errorStatus
              OR runEngine.errorStatus
              OR filling.errorStatus;

  StrAlg.Top:=   runOilsystem.topStatus
              OR runEngine.topStatus
              OR filling.topStatus;

  (*TODO: TYPE PROGRAM CODE HERE*)
  StrAlg.status :=  SHL(BYTE_TO_DWORD(source_for_Status), 29)
  			OR SHL(BYTE_TO_DWORD(cmd_for_Status), 26)
  			OR SHL(BYTE_TO_DWORD(command_error_for_Status), 23)
  			OR SHL(BOOL_TO_DWORD(StrAlg.OpcCommandsDisabled ), 21)
  			OR SHL(BOOL_TO_DWORD(StrAlg.hasError),4)
  			OR SHL(BOOL_TO_DWORD(StrAlg.CanRun),2)
  			OR SHL(BOOL_TO_DWORD(StrAlg.isEnded),1)
  			OR BOOL_TO_DWORD(StrAlg.isRuning);
END_FUNCTION_BLOCK

FUNCTION_BLOCK Pusk_first_faza1
  VAR_IN_OUT
    StrAlg : struct_Alg;
  END_VAR
  VAR
    timer240 : struct_PhaseAlgoritm;
    pmsMore50 : struct_PhaseAlgoritm;
    pnsOn : struct_PhaseAlgoritm;
    pmsMore300 : struct_PhaseAlgoritm;
    Protection_Pms : struct_PhaseAlgoritm;
    Error_Alg : struct_PhaseAlgoritm;
    fb_timer240 : fb_ph_Timer;
    fb_PnmMore50 : fb_ph_algoritm;
    fb_PnsOn : fb_ph_Switch;
    fb_PmsMore300 : fb_ph_algoritm;
    fb_Protection_Pms : fb_ph_algoritm;
    fb_Error_Alg : fb_ph_algoritm;
    _sunpackerCommand : fb_sunpackerCommand;
    _PhaseAlgoritmAction : TYPE_PhaseAlgoritmAction;
    _statusDualInput : TYPE_statusDualInput;
    _Answers : TYPE_Answers;
    source : BYTE;
    cmd : BYTE;
    lastCmd : BYTE;
    source_for_Status : BYTE;
    cmd_for_Status : BYTE;
    command_error_for_Status : BYTE;
    resetCmdTimer : TON;
    resetCmdTimerPriznak : BOOL;
    onInit : BOOL;
    waitReset : TON;
  END_VAR
  VAR_EXTERNAL
    ModeGpa : TYPE_ModeGpa;
    algManager : struct_AlgoritmsManager;
    IM : ImConfig;
    protections : ProtectionsConfig;
  END_VAR
  VAR
    _statusAi : TYPE_StatusAi;
  END_VAR
  VAR_EXTERNAL
    ai : AiConfig;
  END_VAR

  IF NOT onInit THEN

           fb_timer240(phaseNumber:=0, delay:=T#240S);
           fb_PnmMore50(phaseNumber:=1);
           fb_PnsOn(phaseNumber:=2, act:=_on);
           fb_PmsMore300(phaseNumber:=3);
           fb_Protection_Pms(phaseNumber:=4);
           fb_Error_Alg(phaseNumber:=5);

  onInit:=TRUE;
  END_IF;

  fb_timer240(StrPh:=timer240);
  fb_PnmMore50(StrPh:=pmsMore50);
  fb_PnsOn(StrPh:=pnsOn, IM := Im.pns);
  fb_PmsMore300(StrPh:=pmsMore300);
  fb_Protection_Pms(StrPh:=Protection_Pms);
  fb_Error_Alg(StrPh:=Error_Alg);

  StrAlg.CanRun := StrAlg.inCanRun;
  StrAlg.OpcCommandsDisabled := StrAlg.inOpcCommandsDisabled;

  IF StrAlg.isRuning THEN

      StrAlg.hasError := pnsOn.error;

      (* не взведены защиты - запуск таймера *)
      IF NOT Protection_Pms.top THEN
  	runPhase(timer240);
      END_IF;

      (* не начался запуск пнс - запуск пнс *)
      IF NOT pnsOn.start THEN
  	runPhase(pnsOn);
      END_IF;

      (* запуск пнс завершен - запус защит *)
      IF pnsOn.top THEN
           runPhase(pmsMore50);
           runPhase(pmsMore300);
      END_IF;

      (* не завершился запуск защиты 50 - проверка давления 50 *)
      IF pmsMore50.start AND (NOT pmsMore50.top) THEN
  	IF ai.Pmaslo_sm_nizkoe.interval = _statusAi.NORMAL AND ai.Pmaslo_sm_nizkoe.value > 50.0  THEN
  	   pmsMore50.top := TRUE;
            END_IF;
      END_IF;

      (* не завершился запуск защиты 300 - проверка давления 300 *)
      IF  pmsMore300.start AND (NOT pmsMore300.top) THEN
  	IF ai.Pmaslo_sm_vysokoe.interval = _statusAi.NORMAL AND ai.Pmaslo_sm_vysokoe.value > 300.0  THEN
  	    pmsMore300.top := TRUE;
  	END_IF;
      END_IF;

      (* давление было проверено - запуск защит *)
      IF pmsMore50.top AND pmsMore300.top THEN
          runPhase(Protection_Pms);
      END_IF;

      (* запуск защит не завршен - запуск защит *)
      IF Protection_Pms.start AND (NOT Protection_Pms.top) THEN
  	runAiProtection(protections.Pmaslo_sm_nizkoe);
            runAiProtection(protections.Pmaslo_sm_vysokoe);
            Protection_Pms.top := TRUE;
      END_IF;

      (* таймер завершился до запуска защит - ошибка *)
      IF timer240.top THEN
          Error_Alg.ERROR := TRUE; (*не понятное куда его сунуть и нужен ли он*)
      ELSE
          Error_Alg.ERROR := FALSE;
      END_IF;

      (* защиты выствалены до завршения таймера - сброс таймера *)
      IF Protection_Pms.top THEN
  	resetPhase(timer240);
      END_IF;

      StrAlg.isEnded:= pnsOn.Top AND Protection_Pms.Top (*Как будто нужно таймер *);
  END_IF;

  StrAlg.CanRun := StrAlg.inCanRun;
  StrAlg.OpcCommandsDisabled := StrAlg.inOpcCommandsDisabled;

  (* ---- Если управление с ВУ заблокировано, то  передаем команду из алгоритма ---- *)
  IF StrAlg.inOpcCommandsDisabled THEN
  	StrAlg.inCommand := StrAlg.inCommand_Alg;
  ELSE (* иначе передаем команду с АРМа*)
  	StrAlg.inCommand := StrAlg.inCommand_ARM;
  END_IF;

  _sunpackerCommand(command := StrAlg.inCommand);
  	source := _sunpackerCommand.source;
  	cmd := _sunpackerCommand.cmd;

  IF cmd <> 0 AND lastCmd <> cmd AND (((NOT StrAlg.opcCommandsDisabled) AND source > 0) OR source = 0) then
  	CASE BYTE_TO_INT(cmd) OF
  		(*cmdRun*) 1: 	IF (StrAlg.CanRun) THEN
  					StrAlg.isRuning := TRUE;
  					StrAlg.isEnded := FALSE;
  					StrAlg.hasError := FALSE;
  					(*****************       OnRun       *****************)
                                                    algManager.nMode:=ModeGpa.MODE_PUSK_FIRST_FAZA1;

                                                    runPhase(pnsOn);
                                                    resetAiProtection(protections.Pmaslo_sm_nizkoe);
                                                    resetAiProtection(protections.Pmaslo_sm_vysokoe);

  					cmd_for_Status := cmd;
  					source_for_Status := source;
  					command_error_for_Status := 0;
  				ELSE
  					StrAlg.isRuning := FALSE;
  					StrAlg.isEnded := FALSE;
  					StrAlg.hasError := FALSE;

  					cmd_for_Status := 0;
  					source_for_Status := source;
  					command_error_for_Status := cmd;
  				END_IF;
  		(*cmdReset*) 2: 	StrAlg.isRuning := FALSE;
  				StrAlg.isEnded := FALSE;
  				StrAlg.hasError 	:= FALSE;

                                           (*****************       OnReset       *****************)
                                          waitReset(IN:=FALSE);
                                          StrAlg.inCanRun:=FALSE;

                                          resetPhase(timer240);
                                          resetPhase(pmsMore50);
                                          resetPhase(pnsOn);
                                          resetPhase(pmsMore300);
                                          resetPhase(Protection_Pms);
                                          resetPhase(Error_Alg);

                                          StrAlg.inOpcCommandsDisabled:=FALSE;

  				cmd_for_Status := cmd;
  				source_for_Status := source;
  				command_error_for_Status := 0;
  	END_CASE;
  	resetCmdTimer(IN := false);
  	resetCmdTimerPriznak := TRUE;
  END_IF;
  lastCmd := cmd;

  resetCmdTimer(IN := resetCmdTimerPriznak, PT := T#5S);
  IF resetCmdTimer.Q THEN
  	resetCmdTimerPriznak := FALSE;
  	source_for_Status := 0;
  	cmd_for_Status := 0;
  	command_error_for_Status := 0;
  END_IF;

  StrAlg.Start:= timer240.startStatus
              OR pmsMore50.startStatus
              OR pnsOn.startStatus
              OR Error_Alg.startStatus
              OR pmsMore300.startStatus
              OR Protection_Pms.startStatus;

  StrAlg.Error := timer240.errorStatus
              OR pmsMore50.errorStatus
              OR pnsOn.errorStatus
              OR Error_Alg.errorStatus
              OR pmsMore300.errorStatus
              OR Protection_Pms.errorStatus;

  StrAlg.Top := timer240.topStatus
              OR pmsMore50.topStatus
              OR pnsOn.topStatus
              OR Error_Alg.topStatus
              OR pmsMore300.topStatus
              OR Protection_Pms.topStatus;

  (*TODO: TYPE PROGRAM CODE HERE*)
  StrAlg.status :=  SHL(BYTE_TO_DWORD(source_for_Status), 29)
  			OR SHL(BYTE_TO_DWORD(cmd_for_Status), 26)
  			OR SHL(BYTE_TO_DWORD(command_error_for_Status), 23)
  			OR SHL(BOOL_TO_DWORD(StrAlg.OpcCommandsDisabled ), 21)
  			OR SHL(BOOL_TO_DWORD(StrAlg.hasError),4)
  			OR SHL(BOOL_TO_DWORD(StrAlg.CanRun),2)
  			OR SHL(BOOL_TO_DWORD(StrAlg.isEnded),1)
  			OR BOOL_TO_DWORD(StrAlg.isRuning);
END_FUNCTION_BLOCK

FUNCTION_BLOCK Pusk_second_faza_chastotny
  VAR_IN_OUT
    StrAlg : struct_Alg;
  END_VAR
  VAR
    timer120 : struct_PhaseAlgoritm;
    timer5 : struct_PhaseAlgoritm;
    Shup : struct_PhaseAlgoritm;
    Net_Chast : struct_PhaseAlgoritm;
    mvOn : struct_PhaseAlgoritm;
    pGNSmore04 : struct_PhaseAlgoritm;
    gotov_K_zagruzke : struct_PhaseAlgoritm;
    dPmg_Top : struct_PhaseAlgoritm;
    AutoPNS_Start : struct_PhaseAlgoritm;
    fb_timer120 : fb_ph_Timer;
    fb_timer5 : fb_ph_Timer;
    fb_Shup : fb_ph_OilPump;
    fb_Net_Chast : fb_ph_algoritm;
    fb_mvOn : fb_ph_SectionSwitch;
    fb_pGNSmore04 : fb_ph_algoritm;
    fb_gotov_K_zagruzke : fb_ph_algoritm;
    fb_dPmg_Top : fb_ph_algoritm;
    fb_AutoPNS_Start : fb_ph_algoritm;
    _sunpackerCommand : fb_sunpackerCommand;
    _statusDualInput : TYPE_statusDualInput;
    _Answers : TYPE_Answers;
    source : BYTE;
    cmd : BYTE;
    lastCmd : BYTE;
    source_for_Status : BYTE;
    cmd_for_Status : BYTE;
    command_error_for_Status : BYTE;
    resetCmdTimer : TON;
    resetCmdTimerPriznak : BOOL;
    onInit : BOOL;
    waitReset : TON;
  END_VAR
  VAR_EXTERNAL
    ModeGpa : TYPE_ModeGpa;
    algManager : struct_AlgoritmsManager;
    IM : ImConfig;
    protections : ProtectionsConfig;
    algoritms : AlgoritmsConfig;
    ai : AiConfig;
  END_VAR
  VAR
    statusAi : TYPE_StatusAi;
  END_VAR

  IF NOT onInit THEN
           fb_timer120(phaseNumber:=1, delay:=T#120S);
           fb_timer5(phaseNumber:=2, delay:=T#5S);
           fb_Shup(phaseNumber:=3);
           fb_Net_Chast(phaseNumber:=4);
           fb_mvOn(phaseNumber:=5,  act:=_on);
           fb_pGNSmore04(phaseNumber:=6);
           fb_gotov_K_zagruzke(phaseNumber:=7);
           fb_dPmg_Top(phaseNumber:=8);
           fb_AutoPNS_Start(phaseNumber:=9, act:=_run, waitCompletion:=FALSE);
  onInit:=TRUE;
  END_IF;

  fb_timer120(StrPh:=timer120);
  fb_timer5(StrPh:= timer5);
  fb_Shup(StrPh:= Shup);
  fb_Net_Chast(StrPh:=Net_Chast);
  fb_mvOn(StrPh:=mvOn, Im:=IM.mv);
  fb_pGNSmore04(StrPh:=pGNSmore04);
  fb_gotov_K_zagruzke(StrPh:=gotov_K_zagruzke);
  fb_dPmg_Top(StrPh:=dPmg_Top);
  fb_AutoPNS_Start(StrPh:=AutoPNS_Start, alg:=algoritms.autoPns);

  StrAlg.CanRun := StrAlg.inCanRun;
  StrAlg.OpcCommandsDisabled := StrAlg.inOpcCommandsDisabled;

  IF StrAlg.isRuning THEN
      (* мв не включен - запуск таймера *)
      IF NOT mvOn.top THEN
  	runphase(timer120);
      END_IF;
      (* частотный пуск не совершен - запуск таймера *)
      IF NOT Net_Chast.top THEN
  	runphase(timer5);
      END_IF;

      (* ШУП не запущен - запуск *)
      IF NOT Shup.start THEN
  	runphase(Shup);
      END_IF;

      (* ШУП не завершился - запуск ШУПб МВ *)
      IF NOT Shup.top AND Shup.start THEN
  	runIfNotRunningSO(IM.SingleOutputs.Pusk_SHUP);
  	Shup.top:=TRUE;
  	runphase(mvOn);
      END_IF;

      (* частотный пуск не запущен - запуск *)
      IF NOT Net_Chast.start THEN
  	runphase(Net_Chast);
      END_IF;

      (* частотный пуск не завершился - запуск *)
      IF Net_Chast.start AND (NOT Net_Chast.top) THEN
  	IF (NOT IM.SingleSignals.Chastotny_pusk.Q) AND (IM.SingleSignals.Chastotny_pusk.status = 1) THEN
  		Net_Chast.top:=TRUE;
  		resetPhase(timer5);
  	END_IF;
      END_IF;

      (* таймер не истек и мв не включен - вовзедение защиты *)
      IF (NOT timer120.top) AND (NOT mvOn.top) THEN
  	runDiProtection(protections.Fail_chastotnii_pusk);
      ELSE
  	resetDiProtection(protections.Fail_chastotnii_pusk);
      END_IF;

      (* мв не завершился - включение мв *)
      IF mvOn.start AND NOT mvOn.top THEN
  	IF IM.mv.onStatus = _statusDualInput.STATUS_ON THEN
                mvOn.top:=TRUE;
  	END_IF;
      END_IF;

      (* мв завершился - что-то делаем *)
      IF mvOn.top THEN
  	IF NOT pGNSmore04.start (*AND (algManager.mode = ModeGpa.MODE_PUSKPP_Ch OR algManager.mode = ModeGpa.MODE_PUSKAP_Ch)какой режим *) THEN
  		runphase(pGNSmore04);
  	END_IF;
           (* IF NOT autoAVOM_canrun_flag THEN
                algoritms.AutoAvom.CanRun:=TRUE;
  	    autoAVOM_canrun_flag:=TRUE; kto ti
  	END_IF;*)
  	resetPhase(timer120);
  	runphase(gotov_K_zagruzke);

            IF NOT dPmg_Top.start (* AND ((algManager.mode = modegpa.MODE_PUSKAP_Ch) OR (algManager.mode = modegpa.MODE_PUSKPP_Ch))*) THEN
                runphase(dPmg_Top);
  	END_IF;

            runAiProtection(protections.Pgaza_na_vyhode_nagnetatelia_GPA_STOP);
  	runDiProtection(protections.Off_avar_vikluchatel);
  	runDiProtection(protections.Reg_vozb_off);
      END_IF;

      IF dPmg_Top.start AND NOT dPmg_Top.top THEN
  	IF NOT IM.SingleSignals.dP_maslo_gaz_Less100.Q AND IM.SingleSignals.dP_maslo_gaz_Less100.status = 1 AND ai.dPmaslo_gaz.value > 150.0 THEN
  		dPmg_Top.top:=TRUE;
  		runAiProtection(protections.dPmaslo_gaz);
  		runDiProtection(protections.dPmaslo_gaz_less100);
  		resetAiProtection(protections.Pgaza_na_vhode_nagnetatelia_GPA_STOP);
  		resetAiProtection(protections.Pgaza_na_vyhode_nagnetatelia_GPA_STOP);
  		algoritms.autoNu.CanRun:=TRUE;
  		(*algoritms.autoNu.run(); кого чего, ничего не понимаю *)
  	END_IF;
      END_IF;

      IF pGNSmore04.start AND NOT pGNSmore04.top THEN
  	IF ai.Pmasla_posle_GNS.interval (*почему интервал, если есть статус *) >= statusAi.NORMAL AND ai.Pmasla_posle_GNS.value > 400.0 THEN
  	  	pGNSmore04.top:=TRUE;
  	END_IF;
      END_IF;

      IF (pGNSmore04.top AND gotov_K_zagruzke.top AND dPmg_Top.top )(*AND (algManager.mode = modegpa.MODE_PUSKAP_Ch OR (algManager.mode = modegpa.MODE_PUSKPP_Ch) *)OR
  	(gotov_K_zagruzke.top) (*AND (algManager.mode = modegpa.MODE_PUSKV_Ch OR algManager.mode = modegpa.MODE_I))*) AND NOT AutoPNS_Start.top  THEN
  	algoritms.AutoPns.CanRun :=TRUE;
  	(*algoritms.AutoPns;*)
  	AutoPNS_Start.top:=TRUE;
      END_IF;

      IF (NOT Net_Chast.top AND timer5.top) OR (timer120.top AND NOT mvOn.top) THEN
  	algoritms.ao.CanRun:=TRUE;
  	(*algoritms.ao.run ();*)
      END_IF;
  END_IF;

  StrAlg.CanRun := StrAlg.inCanRun;
  StrAlg.OpcCommandsDisabled := StrAlg.inOpcCommandsDisabled;

  (* ---- Если управление с ВУ заблокировано, то  передаем команду из алгоритма ---- *)
  IF StrAlg.inOpcCommandsDisabled THEN
  	StrAlg.inCommand := StrAlg.inCommand_Alg;
  ELSE (* иначе передаем команду с АРМа*)
  	StrAlg.inCommand := StrAlg.inCommand_ARM;
  END_IF;

  _sunpackerCommand(command := StrAlg.inCommand);
  	source := _sunpackerCommand.source;
  	cmd := _sunpackerCommand.cmd;

  IF cmd <> 0 AND lastCmd <> cmd AND (((NOT StrAlg.opcCommandsDisabled) AND source > 0) OR source = 0) then
  	CASE BYTE_TO_INT(cmd) OF
  		(*cmdRun*) 1: 	IF (StrAlg.CanRun) THEN
  					StrAlg.isRuning := TRUE;
  					StrAlg.isEnded := FALSE;
  					StrAlg.hasError := FALSE;
  					(*****************       OnRun       *****************)
                                                    algManager.nMode:=ModeGpa.MODE_PUSK_FIRST_FAZA2;

                                                    runPhase(timer120);
                                                    runPhase(timer5);
                                                    runPhase(Shup);
                                                    resetAiProtection(protections.dPmaslo_gaz);
                                                    resetDiProtection(protections.dPmaslo_gaz_less100);

  					cmd_for_Status := cmd;
  					source_for_Status := source;
  					command_error_for_Status := 0;
  				ELSE
  					StrAlg.isRuning := FALSE;
  					StrAlg.isEnded := FALSE;
  					StrAlg.hasError := FALSE;

  					cmd_for_Status := 0;
  					source_for_Status := source;
  					command_error_for_Status := cmd;
  				END_IF;
  		(*cmdReset*) 2: 	StrAlg.isRuning := FALSE;
  				StrAlg.isEnded := FALSE;
  				StrAlg.hasError 	:= FALSE;

                                           (*****************       OnReset       *****************)
                                          waitReset(IN:=FALSE);
                                          StrAlg.inCanRun:=FALSE;

                                          resetPhase(timer5);
                                          resetPhase(Shup);
                                          resetPhase(timer120);
                                          resetPhase(Net_Chast);
                                          resetPhase(mvOn);
                                          resetPhase(pGNSmore04);
                                          resetPhase(gotov_K_zagruzke);
                                          resetPhase(dPmg_Top);
                                          resetPhase(AutoPNS_Start);

                                          StrAlg.inOpcCommandsDisabled:=FALSE;

  				cmd_for_Status := cmd;
  				source_for_Status := source;
  				command_error_for_Status := 0;
  	END_CASE;
  	resetCmdTimer(IN := false);
  	resetCmdTimerPriznak := TRUE;
  END_IF;
  lastCmd := cmd;

  resetCmdTimer(IN := resetCmdTimerPriznak, PT := T#5S);
  IF resetCmdTimer.Q THEN
  	resetCmdTimerPriznak := FALSE;
  	source_for_Status := 0;
  	cmd_for_Status := 0;
  	command_error_for_Status := 0;
  END_IF;

  StrAlg.Start:= timer120.startStatus
              OR timer5.startStatus
              OR Shup.startStatus
              OR Net_Chast.startStatus
              OR mvOn.startStatus
              OR pGNSmore04.startStatus
              OR gotov_K_zagruzke.startStatus
              OR dPmg_Top.startStatus
              OR AutoPNS_Start.startStatus;

  StrAlg.Error := timer120.errorStatus
              OR timer5.errorStatus
              OR Shup.errorStatus
              OR Net_Chast.errorStatus
              OR mvOn.errorStatus
              OR pGNSmore04.errorStatus
              OR gotov_K_zagruzke.errorStatus
              OR dPmg_Top.errorStatus
              OR AutoPNS_Start.errorStatus;

  StrAlg.Top := timer120.topStatus
              OR timer5.topStatus
              OR Shup.topStatus
              OR Net_Chast.topStatus
              OR mvOn.topStatus
              OR gotov_K_zagruzke.topStatus
              OR dPmg_Top.topStatus
              OR AutoPNS_Start.topStatus
              OR pGNSmore04.topStatus;

  (*TODO: TYPE PROGRAM CODE HERE*)
  StrAlg.status :=  SHL(BYTE_TO_DWORD(source_for_Status), 29)
  			OR SHL(BYTE_TO_DWORD(cmd_for_Status), 26)
  			OR SHL(BYTE_TO_DWORD(command_error_for_Status), 23)
  			OR SHL(BOOL_TO_DWORD(StrAlg.OpcCommandsDisabled ), 21)
  			OR SHL(BOOL_TO_DWORD(StrAlg.hasError),4)
  			OR SHL(BOOL_TO_DWORD(StrAlg.CanRun),2)
  			OR SHL(BOOL_TO_DWORD(StrAlg.isEnded),1)
  			OR BOOL_TO_DWORD(StrAlg.isRuning);
END_FUNCTION_BLOCK

FUNCTION_BLOCK proc_algoritms
  VAR
    fb_RemontAlg : RemontAlg;
    fb_TestProtectionAlg : TestProtectionAlg;
    fb_TestImAlg : TestImAlg;
    fb_AutoTen : fb_AutoTenAlg;
    fb_AutoPns : fb_AutoPnsAlg;
    fb_AutoAvom : fb_AutoAvomAlg;
    fb_vibegPNS : fb_vibegPNSAlg;
    fb_AutoNU : fb_AutoNUAlg;
    fb_puskOilSystem : fb_puskOilSystemAlg;
    fb_AntiPompag : fb_AntiPompagAlg;
    fb_NOAlg : NOAlg;
    fb_AOAlg : AOAlg;
    fb_ppuALG : ppuAlg;
    fb_fillingAlg : fillingAlg;
    fb_engineRunAlg : engineRunAlg;
    fb_puskKalg : puskKalg;
    fb_puskValg : puskValg;
    fb_testdPmgAlg : testdPmgAlg;
    fb_testPmsAlg : testPmsAlg;
    fb_ApuskAlg : ApuskAlg;
    fb_SemiAutoPuskAlg : SemiAutoPuskAlg;
    fb_Pusk_first_faza1 : Pusk_first_faza1;
    fb_Pusk_first_faza2 : Pusk_first_faza2;
    fb_Pusk_third_faza : Pusk_third_faza;
    fb_Pusk_Prov_PMS : Prov_PMS;
    fb_Prov_opressovka : Prov_opressovka;
    fb_Pusk_second_faza_chastotny : Pusk_second_faza_chastotny;
    fb_Pusk_second_faza_reactor : Pusk_second_faza_reactor;
  END_VAR
  VAR_EXTERNAL
    algoritms : AlgoritmsConfig;
    AlgQuestions : AlgoritmsQuestions;
    ai : AiConfig;
    IM : ImConfig;
    AlgTimers : struct_AlgTimers;
  END_VAR

  fb_RemontAlg(StrAlg:=algoritms.Remont);

  fb_TestProtectionAlg(StrAlg:=algoritms.TestProtection);

  fb_TestImAlg(StrAlg:=algoritms.testIm);

  (*fb_AutoTen(StrAlg:= algoritms.AutoTen,
  T_masla:= ai.Toporno_podshipnika_EDT_1,
  Uroven_masla:= ai.Yroven_masla_MB,
  offTemperature:= Im.AutoTen_offTemperature,
  TEN:= Im.Ten,
  PNS:= Im.pns);*)

  (*fb_AutoPns(StrAlg:= algoritms.AutoPns,
  Poil:= ai.Pmasla_posle_GNS,
  Ust_Run:= Im.AutoPns_UstRun,
  Ust_Stop:= Im.AutoPns_UstStop,
  Nasos:= Im.pns,
  diPlow:= Im.SingleSignals.P_oil_low);*)

  (*fb_AutoAvom(StrAlg:= algoritms.AutoAvom,
  im1:= Im.v1_Avom,
  im2:= Im.v2_Avom,
  on1Temperature:= Im.AutoAvom_onTemp1,
  on2Temperature:= Im.AutoAvom_onTemp2,
  hystereses:= Im.AutoAvom_hysteresis,
  ai:= ai.Tnarujnogo_vozduha);*)

  fb_vibegPNS(StrAlg:=algoritms.vibegPNS,
  algContinue:=AlgQuestions.vibegPNS_algContinue
  );

  (*fb_AutoNU(StrAlg:=algoritms.autoNu,
  nu1:=Im.nu1,
  nu2:=Im.nu2,
  Ust_Swap:= Im.AutoNU_Ust_Swap,
  mainNU:= Im.AutoNU_mainNU,
  dPoil:=ai.Tmasla_MB,
  Lowdp_di:=Im.SingleSignals.dP_oilgaz_low
  );*)

  fb_puskOilSystem(StrAlg:=algoritms.puskOilSystem);

  (*fb_AntiPompag(StrAlg:=algoritms.AntiPompag,
  Rashod:= ai.Vibro_skorost_OP_shesterni_RED_T6,
  Zapas:= ai.Vibro_skorost_OP_shesterni_RED_T5,
  P_gasIn:=ai.dPgaza_na_maslo_filtre,
  T_gasIn:=ai.Tgaza_na_vhode_H,
  dP_konf:=ai.dPgaza_na_konfuzore,
  Kran6:= im.Kran6,
  UgolVNA:= im.AntiPompag_UgolVNA,
  K:=im.AntiPompag_K,
  A:=im.AntiPompag_A,
  y0:=im.AntiPompag_y0);*)

  fb_NOAlg(StrAlg:=algoritms.no);

  fb_AOAlg(StrAlg:=algoritms.ao);

  fb_ppuAlg(StrAlg:=algoritms.ppu);

  fb_fillingAlg(StrAlg:=algoritms.filling);

  fb_engineRunAlg(StrAlg:=algoritms.engineRun);

  fb_puskKalg(StrAlg:=algoritms.puskK,
  questionFilling:=AlgQuestions.puskK_questionFilling,
   questionUnload:=AlgQuestions.puskK_questionUnload
  );

  fb_puskValg(StrAlg:=algoritms.puskV,
   questionEngine:=AlgQuestions.puskV_questionEngine,
    questionMVoff:=AlgQuestions.puskV_questionMVoff
  );

  fb_testdPmgAlg(StrAlg:=algoritms.testdPmg,
   algContinue:=AlgQuestions.testdPmg_algContinue
  );

  fb_testPmsAlg(StrAlg:=algoritms.testPms,
   algContinue:=AlgQuestions.testPms_algContinue
  );

  fb_ApuskAlg(StrAlg:=algoritms.Apusk);

  fb_SemiAutoPuskAlg(StrAlg:=algoritms.SemiAutoPusk,
   cmdRun1ph:=AlgQuestions.SemiAutoPusk_cmdRun1ph,
   cmdRun2ph:=AlgQuestions.SemiAutoPusk_cmdRun2ph,
   cmdRun3ph:=AlgQuestions.SemiAutoPusk_cmdRun3ph
  );

  fb_Pusk_first_faza1(Stralg:=algoritms.Pusk_F_faza1);

  fb_Pusk_first_faza2(Stralg:=algoritms.Pusk_F_faza2);

  fb_Pusk_third_faza(Stralg:=algoritms.Pusk_TH_faza);

  fb_Pusk_Prov_PMS(Stralg:=algoritms.Prov_PMS_ALG);

  fb_Prov_opressovka(Stralg:=algoritms.Prov_opressovka_ALG);

  fb_Pusk_second_faza_chastotny(Stralg:=algoritms.Pusk_SEC_faza_chastotny);

  fb_Pusk_second_faza_reactor(Stralg:=algoritms.Pusk_SEC_faza_reactor);
END_FUNCTION_BLOCK

FUNCTION_BLOCK proc_AI_Init
  VAR_INPUT
    init : BOOL;
  END_VAR
  VAR
    stAI_Ini : fb_AI_Init;
    inits : UINT;
  END_VAR
  VAR_INPUT
    initiales : UINT;
  END_VAR
  VAR_EXTERNAL
    ai : AiConfig;
  END_VAR

  inits := 0; (* Флаг необходимости инициализации структур-дескрипторов *)

  (********************************************* Модуль A2-14 ******************************************************)
  (* [A2-14, AI0-0] TStalisStatoraKanal1 *)
  stAI_Ini(data_Ini := TRUE, dLL := 0.0, dHL := 150.0,
  ISVALIDREF_HW := TRUE, dHW := 130.0, aperturFilter:= 0.5,
  strAI := ai.Tstali_statora_kanal_1);
  inits := inits + BOOL_TO_UINT(stAI_Ini.Init);

  (* [A2-14, AI0-1] TStalisStatoraKanal2 *)
  stAI_Ini(data_Ini := TRUE,  dLL := 0.0, dHL := 150.0,
  ISVALIDREF_HW := TRUE, dHW := 130.0, aperturFilter:= 0.5,
  strAI := ai.Tstali_statora_kanal_2);
  inits := inits + BOOL_TO_UINT(stAI_Ini.Init);

  (* [A2-14, AI0-2] TStalisStatoraKanal3 *)
  stAI_Ini(data_Ini := TRUE,  dLL := 0.0, dHL :=150.0,
  ISVALIDREF_HW := TRUE, dHW := 130.0, aperturFilter:= 0.5,
  strAI := ai.Tstali_statora_kanal_3);
  inits := inits + BOOL_TO_UINT(stAI_Ini.Init);

  (* [A2-14, AI0-3] TMediStatoraKanal1 *)
  stAI_Ini(data_Ini := TRUE,  dLL := 0.0, dHL := 150.0,
  ISVALIDREF_HW := TRUE, dHW := 130.0, aperturFilter:= 0.5,
  strAI := ai.Tmedi_statora_kanal_1);
  inits := inits + BOOL_TO_UINT(stAI_Ini.Init);

  (********************************************* Модуль A2-15 ******************************************************)

  (* [A2-15, AI1-0] TMediStatoraKanal2 *)
  stAI_Ini(data_Ini :=TRUE,  dLL := 0.0, dHL := 150.0,
  ISVALIDREF_HW := TRUE, dHW := 130.0, aperturFilter:= 0.5,
  strAI := ai.Tmedi_statora_kanal_2);
  inits := inits + BOOL_TO_UINT(stAI_Ini.Init);

  (* [A2-15, AI1-1] TMediStatoraKanal3 *)
  stAI_Ini(data_Ini := TRUE,  dLL := 0.0, dHL := 150.0,
  ISVALIDREF_HW := TRUE, dHW := 130.0, aperturFilter:= 0.5,
  strAI := ai.Tmedi_statora_kanal_3);
  inits := inits + BOOL_TO_UINT(stAI_Ini.Init);

  (* [A2-15, AI1-2] TOpornogoPodshipnikaEDT_1 *)
  stAI_Ini(data_Ini := TRUE,  dLL := 0.0, dHL := 100.0,
  ISVALIDREF_HA := TRUE, ISVALIDREF_HW := TRUE, dHA := 80.0, dHW := 75.0, aperturFilter:= 0.5, dMaxChangeSpeed := 10.0,
  strAI := ai.Toporno_podshipnika_EDT_1);
  inits := inits + BOOL_TO_UINT(stAI_Ini.Init);
